//     Enc/Inputs/In/nState2 @bit 1 <-> ENC Status compact/Status/Status of input B
//     Enc/Inputs/In/nState2 @bit 2 <-> ENC Status compact/Status/Status of input C
//     Enc/Inputs/In/nState2 @bit 5 <-> ENC Status compact/Status/Sync error
//     Enc/Inputs/In/nState2 @bit 7 <-> ENC Status compact/Status/TxPDO Toggle
//     Enc/Inputs/In/nState4 @bit 1 <-> WcState/InputToggle
//     Enc/Inputs/In/nState4 <-> WcState/WcState
//     Enc/Outputs/Out/nCtrl1 <-> ENC Control compact/Control/Enable latch C
//     Enc/Outputs/Out/nCtrl1 @bit 3 <-> ENC Control compact/Control/Enable latch extern on negative edge
//     Enc/Outputs/Out/nCtrl1 @bit 1 <-> ENC Control compact/Control/Enable latch extern on positive edge
//     Enc/Outputs/Out/nCtrl1 @bit 2 <-> ENC Control compact/Control/Set counter
//     Enc/Outputs/Out/nDataOut1[0] <-> ENC Control compact/Set counter value
//   (this object) <-> Device 1 (EtherCAT)/Term 5 (EK1200)/Term 6 (EK1122-0080)/DRL02-EK0 (EK1101-0080)/DRL02-E21 (EL7041)
//     Drive/Inputs/In/nState1 @bit 3 <-> STM Status/Status/Error
//     Drive/Inputs/In/nState1 @bit 5 <-> STM Status/Status/Moving negative
//     Drive/Inputs/In/nState1 @bit 4 <-> STM Status/Status/Moving positive
//     Drive/Inputs/In/nState1 @bit 1 <-> STM Status/Status/Ready
//     Drive/Inputs/In/nState1 <-> STM Status/Status/Ready to enable
//     Drive/Inputs/In/nState1 @bit 6 <-> STM Status/Status/Torque reduced
//     Drive/Inputs/In/nState1 @bit 2 <-> STM Status/Status/Warning
//     Drive/Inputs/In/nState2 @bit 3 <-> STM Status/Status/Digital input 1
//     Drive/Inputs/In/nState2 @bit 4 <-> STM Status/Status/Digital input 2
//     Drive/Inputs/In/nState2 @bit 5 <-> STM Status/Status/Sync error
//     Drive/Inputs/In/nState2 @bit 7 <-> STM Status/Status/TxPDO Toggle
//     Drive/Inputs/In/nState4 @bit 1 <-> WcState/InputToggle
//     Drive/Inputs/In/nState4 <-> WcState/WcState
//     Drive/Outputs/Out/nCtrl1 <-> STM Control/Control/Enable
//     Drive/Outputs/Out/nCtrl1 @bit 2 <-> STM Control/Control/Reduce torque
//     Drive/Outputs/Out/nCtrl1 @bit 1 <-> STM Control/Control/Reset
//     Drive/Outputs/Out/nDataOut2[0] <-> STM Velocity/Velocity
//     Enc/Inputs/In/nDataIn1[0] <-> ENC Status compact/Counter value
//     Enc/Inputs/In/nDataIn2[0] <-> ENC Status compact/Latch value
//     Enc/Inputs/In/nState1 @bit 4 <-> ENC Status compact/Status/Counter overflow
//     Enc/Inputs/In/nState1 @bit 3 <-> ENC Status compact/Status/Counter underflow
//     Enc/Inputs/In/nState1 @bit 7 <-> ENC Status compact/Status/Extrapolation stall
//     Enc/Inputs/In/nState1 <-> ENC Status compact/Status/Latch C valid
//     Enc/Inputs/In/nState1 @bit 1 <-> ENC Status compact/Status/Latch extern valid
//     Enc/Inputs/In/nState1 @bit 2 <-> ENC Status compact/Status/Set counter done
//     Enc/Inputs/In/nState2 @bit 4 <-> ENC Status compact/Status/Status of extern latch
//     Enc/Inputs/In/nState2 <-> ENC Status compact/Status/Status of input A
//     Enc/Inputs/In/nState2 @bit 1 <-> ENC Status compact/Status/Status of input B
//     Enc/Inputs/In/nState2 @bit 2 <-> ENC Status compact/Status/Status of input C
//     Enc/Inputs/In/nState2 @bit 5 <-> ENC Status compact/Status/Sync error
//     Enc/Inputs/In/nState2 @bit 7 <-> ENC Status compact/Status/TxPDO Toggle
//     Enc/Inputs/In/nState4 @bit 1 <-> WcState/InputToggle
//     Enc/Inputs/In/nState4 <-> WcState/WcState
//     Enc/Outputs/Out/nCtrl1 <-> ENC Control compact/Control/Enable latch C
//     Enc/Outputs/Out/nCtrl1 @bit 3 <-> ENC Control compact/Control/Enable latch extern on negative edge
//     Enc/Outputs/Out/nCtrl1 @bit 1 <-> ENC Control compact/Control/Enable latch extern on positive edge
//     Enc/Outputs/Out/nCtrl1 @bit 2 <-> ENC Control compact/Control/Set counter
//     Enc/Outputs/Out/nDataOut1[0] <-> ENC Control compact/Set counter value
//   (this object) <-> Device 1 (EtherCAT)/Term 5 (EK1200)/Term 6 (EK1122-0080)/DRL02-EK0 (EK1101-0080)/DRL02-E1 (EL7031)
//     Drive/Inputs/In/nState1 @bit 3 <-> STM Status/Status/Error
//     Drive/Inputs/In/nState1 @bit 5 <-> STM Status/Status/Moving negative
//     Drive/Inputs/In/nState1 @bit 4 <-> STM Status/Status/Moving positive
//     Drive/Inputs/In/nState1 @bit 1 <-> STM Status/Status/Ready
//     Drive/Inputs/In/nState1 <-> STM Status/Status/Ready to enable
//     Drive/Inputs/In/nState1 @bit 6 <-> STM Status/Status/Torque reduced
//     Drive/Inputs/In/nState1 @bit 2 <-> STM Status/Status/Warning
//     Drive/Inputs/In/nState2 @bit 3 <-> STM Status/Status/Digital input 1
//     Drive/Inputs/In/nState2 @bit 4 <-> STM Status/Status/Digital input 2
//     Drive/Inputs/In/nState2 @bit 5 <-> STM Status/Status/Sync error
//     Drive/Inputs/In/nState2 @bit 7 <-> STM Status/Status/TxPDO Toggle
//     Drive/Inputs/In/nState4 @bit 1 <-> WcState/InputToggle
//     Drive/Inputs/In/nState4 <-> WcState/WcState
//     Drive/Outputs/Out/nCtrl1 <-> STM Control/Control/Enable
//     Drive/Outputs/Out/nCtrl1 @bit 2 <-> STM Control/Control/Reduce torque
//     Drive/Outputs/Out/nCtrl1 @bit 1 <-> STM Control/Control/Reset
//     Drive/Outputs/Out/nDataOut2[0] <-> STM Velocity/Velocity
//   (this object) <-> Device 1 (EtherCAT)/Term 5 (EK1200)/Term 6 (EK1122-0080)/DRL02-EK0 (EK1101-0080)/DRL02-E2 (EL5042)
//     Enc/Inputs/In/nComState @bit 1 <-> WcState/InputToggle
//     Enc/Inputs/In/nComState <-> WcState/WcState
//     Enc/Inputs/In/nDataIn1 <-> FB Inputs Channel 1/Position
//     Enc/Inputs/In/nDataIn1 <-> FB Inputs Channel 2/Position
//     Enc/Inputs/In/nState1 @bit 12 <-> FB Inputs Channel 1/Status/Diag
//     Enc/Inputs/In/nState1 @bit 12 <-> FB Inputs Channel 2/Status/Diag
//     Enc/Inputs/In/nState1 @bit 1 <-> FB Inputs Channel 1/Status/Error
//     Enc/Inputs/In/nState1 @bit 1 <-> FB Inputs Channel 2/Status/Error
//     Enc/Inputs/In/nState1 @bit 14 <-> FB Inputs Channel 1/Status/Input cycle counter
//     Enc/Inputs/In/nState1 @bit 14 <-> FB Inputs Channel 2/Status/Input cycle counter
//     Enc/Inputs/In/nState1 @bit 2 <-> FB Inputs Channel 1/Status/Ready
//     Enc/Inputs/In/nState1 @bit 2 <-> FB Inputs Channel 2/Status/Ready
//     Enc/Inputs/In/nState1 @bit 13 <-> FB Inputs Channel 1/Status/TxPDO State
//     Enc/Inputs/In/nState1 @bit 13 <-> FB Inputs Channel 2/Status/TxPDO State
//     Enc/Inputs/In/nState1 <-> FB Inputs Channel 1/Status/Warning
//     Enc/Inputs/In/nState1 <-> FB Inputs Channel 2/Status/Warning
//   (this object) <-> Device 1 (EtherCAT)/Term 5 (EK1200)/Term 6 (EK1122-0080)/DRL02-EK0 (EK1101-0080)/DRL02-E3 (EL7031)
//     Drive/Inputs/In/nState1 @bit 3 <-> STM Status/Status/Error
//     Drive/Inputs/In/nState1 @bit 5 <-> STM Status/Status/Moving negative
//     Drive/Inputs/In/nState1 @bit 4 <-> STM Status/Status/Moving positive
//     Drive/Inputs/In/nState1 @bit 1 <-> STM Status/Status/Ready
//     Drive/Inputs/In/nState1 <-> STM Status/Status/Ready to enable
//     Drive/Inputs/In/nState1 @bit 6 <-> STM Status/Status/Torque reduced
//     Drive/Inputs/In/nState1 @bit 2 <-> STM Status/Status/Warning
//     Drive/Inputs/In/nState2 @bit 3 <-> STM Status/Status/Digital input 1
//     Drive/Inputs/In/nState2 @bit 4 <-> STM Status/Status/Digital input 2
//     Drive/Inputs/In/nState2 @bit 5 <-> STM Status/Status/Sync error
//     Drive/Inputs/In/nState2 @bit 7 <-> STM Status/Status/TxPDO Toggle
//     Drive/Inputs/In/nState4 @bit 1 <-> WcState/InputToggle
//     Drive/Inputs/In/nState4 <-> WcState/WcState
//     Drive/Outputs/Out/nCtrl1 <-> STM Control/Control/Enable
//     Drive/Outputs/Out/nCtrl1 @bit 2 <-> STM Control/Control/Reduce torque
//     Drive/Outputs/Out/nCtrl1 @bit 1 <-> STM Control/Control/Reset
//     Drive/Outputs/Out/nDataOut2[0] <-> STM Velocity/Velocity
//   (this object) <-> Device 1 (EtherCAT)/Term 5 (EK1200)/Term 6 (EK1122-0080)/DRL02-EK0 (EK1101-0080)/DRL02-E4 (EL7031)
//     Drive/Inputs/In/nState1 @bit 3 <-> STM Status/Status/Error
//     Drive/Inputs/In/nState1 @bit 5 <-> STM Status/Status/Moving negative
//     Drive/Inputs/In/nState1 @bit 4 <-> STM Status/Status/Moving positive
//     Drive/Inputs/In/nState1 @bit 1 <-> STM Status/Status/Ready
//     Drive/Inputs/In/nState1 <-> STM Status/Status/Ready to enable
//     Drive/Inputs/In/nState1 @bit 6 <-> STM Status/Status/Torque reduced
//     Drive/Inputs/In/nState1 @bit 2 <-> STM Status/Status/Warning
//     Drive/Inputs/In/nState2 @bit 3 <-> STM Status/Status/Digital input 1
//     Drive/Inputs/In/nState2 @bit 4 <-> STM Status/Status/Digital input 2
//     Drive/Inputs/In/nState2 @bit 5 <-> STM Status/Status/Sync error
//     Drive/Inputs/In/nState2 @bit 7 <-> STM Status/Status/TxPDO Toggle
//     Drive/Inputs/In/nState4 @bit 1 <-> WcState/InputToggle
//     Drive/Inputs/In/nState4 <-> WcState/WcState
//     Drive/Outputs/Out/nCtrl1 <-> STM Control/Control/Enable
//     Drive/Outputs/Out/nCtrl1 @bit 2 <-> STM Control/Control/Reduce torque
//     Drive/Outputs/Out/nCtrl1 @bit 1 <-> STM Control/Control/Reset
//     Drive/Outputs/Out/nDataOut2[0] <-> STM Velocity/Velocity
//   (this object) <-> Device 1 (EtherCAT)/Term 5 (EK1200)/Term 6 (EK1122-0080)/DRL02-EK0 (EK1101-0080)/DRL02-E5 (EL5042)
//     Enc/Inputs/In/nComState @bit 1 <-> WcState/InputToggle
//     Enc/Inputs/In/nComState <-> WcState/WcState
//     Enc/Inputs/In/nDataIn1 <-> FB Inputs Channel 1/Position
//     Enc/Inputs/In/nDataIn1 <-> FB Inputs Channel 2/Position
//     Enc/Inputs/In/nState1 @bit 12 <-> FB Inputs Channel 1/Status/Diag
//     Enc/Inputs/In/nState1 @bit 12 <-> FB Inputs Channel 2/Status/Diag
//     Enc/Inputs/In/nState1 @bit 1 <-> FB Inputs Channel 1/Status/Error
//     Enc/Inputs/In/nState1 @bit 1 <-> FB Inputs Channel 2/Status/Error
//     Enc/Inputs/In/nState1 @bit 14 <-> FB Inputs Channel 1/Status/Input cycle counter
//     Enc/Inputs/In/nState1 @bit 14 <-> FB Inputs Channel 2/Status/Input cycle counter
//     Enc/Inputs/In/nState1 @bit 2 <-> FB Inputs Channel 1/Status/Ready
//     Enc/Inputs/In/nState1 @bit 2 <-> FB Inputs Channel 2/Status/Ready
//     Enc/Inputs/In/nState1 @bit 13 <-> FB Inputs Channel 1/Status/TxPDO State
//     Enc/Inputs/In/nState1 @bit 13 <-> FB Inputs Channel 2/Status/TxPDO State
//     Enc/Inputs/In/nState1 <-> FB Inputs Channel 1/Status/Warning
//     Enc/Inputs/In/nState1 <-> FB Inputs Channel 2/Status/Warning
//   (this object) <-> Device 1 (EtherCAT)/Term 5 (EK1200)/Term 6 (EK1122-0080)/DRL02-EK0 (EK1101-0080)/DRL02-E6 (EL7031)
//     Drive/Inputs/In/nState1 @bit 3 <-> STM Status/Status/Error
//     Drive/Inputs/In/nState1 @bit 5 <-> STM Status/Status/Moving negative
//     Drive/Inputs/In/nState1 @bit 4 <-> STM Status/Status/Moving positive
//     Drive/Inputs/In/nState1 @bit 1 <-> STM Status/Status/Ready
//     Drive/Inputs/In/nState1 <-> STM Status/Status/Ready to enable
//     Drive/Inputs/In/nState1 @bit 6 <-> STM Status/Status/Torque reduced
//     Drive/Inputs/In/nState1 @bit 2 <-> STM Status/Status/Warning
//     Drive/Inputs/In/nState2 @bit 3 <-> STM Status/Status/Digital input 1
//     Drive/Inputs/In/nState2 @bit 4 <-> STM Status/Status/Digital input 2
//     Drive/Inputs/In/nState2 @bit 5 <-> STM Status/Status/Sync error
//     Drive/Inputs/In/nState2 @bit 7 <-> STM Status/Status/TxPDO Toggle
//     Drive/Inputs/In/nState4 @bit 1 <-> WcState/InputToggle
//     Drive/Inputs/In/nState4 <-> WcState/WcState
//     Drive/Outputs/Out/nCtrl1 <-> STM Control/Control/Enable
//     Drive/Outputs/Out/nCtrl1 @bit 2 <-> STM Control/Control/Reduce torque
//     Drive/Outputs/Out/nCtrl1 @bit 1 <-> STM Control/Control/Reset
//     Drive/Outputs/Out/nDataOut2[0] <-> STM Velocity/Velocity
//   (this object) <-> Device 1 (EtherCAT)/Term 5 (EK1200)/Term 6 (EK1122-0080)/DRL02-EK0 (EK1101-0080)/DRL02-E7 (EL7031)
//     Drive/Inputs/In/nState1 @bit 3 <-> STM Status/Status/Error
//     Drive/Inputs/In/nState1 @bit 5 <-> STM Status/Status/Moving negative
//     Drive/Inputs/In/nState1 @bit 4 <-> STM Status/Status/Moving positive
//     Drive/Inputs/In/nState1 @bit 1 <-> STM Status/Status/Ready
//     Drive/Inputs/In/nState1 <-> STM Status/Status/Ready to enable
//     Drive/Inputs/In/nState1 @bit 6 <-> STM Status/Status/Torque reduced
//     Drive/Inputs/In/nState1 @bit 2 <-> STM Status/Status/Warning
//     Drive/Inputs/In/nState2 @bit 3 <-> STM Status/Status/Digital input 1
//     Drive/Inputs/In/nState2 @bit 4 <-> STM Status/Status/Digital input 2
//     Drive/Inputs/In/nState2 @bit 5 <-> STM Status/Status/Sync error
//     Drive/Inputs/In/nState2 @bit 7 <-> STM Status/Status/TxPDO Toggle
//     Drive/Inputs/In/nState4 @bit 1 <-> WcState/InputToggle
//     Drive/Inputs/In/nState4 <-> WcState/WcState
//     Drive/Outputs/Out/nCtrl1 <-> STM Control/Control/Enable
//     Drive/Outputs/Out/nCtrl1 @bit 2 <-> STM Control/Control/Reduce torque
//     Drive/Outputs/Out/nCtrl1 @bit 1 <-> STM Control/Control/Reset
//     Drive/Outputs/Out/nDataOut2[0] <-> STM Velocity/Velocity
//   (this object) <-> Device 1 (EtherCAT)/Term 5 (EK1200)/Term 6 (EK1122-0080)/DRL02-EK0 (EK1101-0080)/DRL02-E8 (EL5042)
//     Enc/Inputs/In/nComState @bit 1 <-> WcState/InputToggle
//     Enc/Inputs/In/nComState <-> WcState/WcState
//     Enc/Inputs/In/nDataIn1 <-> FB Inputs Channel 1/Position
//     Enc/Inputs/In/nDataIn1 <-> FB Inputs Channel 2/Position
//     Enc/Inputs/In/nState1 @bit 12 <-> FB Inputs Channel 1/Status/Diag
//     Enc/Inputs/In/nState1 @bit 12 <-> FB Inputs Channel 2/Status/Diag
//     Enc/Inputs/In/nState1 @bit 1 <-> FB Inputs Channel 1/Status/Error
//     Enc/Inputs/In/nState1 @bit 1 <-> FB Inputs Channel 2/Status/Error
//     Enc/Inputs/In/nState1 @bit 14 <-> FB Inputs Channel 1/Status/Input cycle counter
//     Enc/Inputs/In/nState1 @bit 14 <-> FB Inputs Channel 2/Status/Input cycle counter
//     Enc/Inputs/In/nState1 @bit 2 <-> FB Inputs Channel 1/Status/Ready
//     Enc/Inputs/In/nState1 @bit 2 <-> FB Inputs Channel 2/Status/Ready
//     Enc/Inputs/In/nState1 @bit 13 <-> FB Inputs Channel 1/Status/TxPDO State
//     Enc/Inputs/In/nState1 @bit 13 <-> FB Inputs Channel 2/Status/TxPDO State
//     Enc/Inputs/In/nState1 <-> FB Inputs Channel 1/Status/Warning
//     Enc/Inputs/In/nState1 <-> FB Inputs Channel 2/Status/Warning
//   (this object) <-> Device 1 (EtherCAT)/Term 5 (EK1200)/Term 6 (EK1122-0080)/DRL02-EK0 (EK1101-0080)/DRL02-E9 (EL7031)
//     Drive/Inputs/In/nState1 @bit 3 <-> STM Status/Status/Error
//     Drive/Inputs/In/nState1 @bit 5 <-> STM Status/Status/Moving negative
//     Drive/Inputs/In/nState1 @bit 4 <-> STM Status/Status/Moving positive
//     Drive/Inputs/In/nState1 @bit 1 <-> STM Status/Status/Ready
//     Drive/Inputs/In/nState1 <-> STM Status/Status/Ready to enable
//     Drive/Inputs/In/nState1 @bit 6 <-> STM Status/Status/Torque reduced
//     Drive/Inputs/In/nState1 @bit 2 <-> STM Status/Status/Warning
//     Drive/Inputs/In/nState2 @bit 3 <-> STM Status/Status/Digital input 1
//     Drive/Inputs/In/nState2 @bit 4 <-> STM Status/Status/Digital input 2
//     Drive/Inputs/In/nState2 @bit 5 <-> STM Status/Status/Sync error
//     Drive/Inputs/In/nState2 @bit 7 <-> STM Status/Status/TxPDO Toggle
//     Drive/Inputs/In/nState4 @bit 1 <-> WcState/InputToggle
//     Drive/Inputs/In/nState4 <-> WcState/WcState
//     Drive/Outputs/Out/nCtrl1 <-> STM Control/Control/Enable
//     Drive/Outputs/Out/nCtrl1 @bit 2 <-> STM Control/Control/Reduce torque
//     Drive/Outputs/Out/nCtrl1 @bit 1 <-> STM Control/Control/Reset
//     Drive/Outputs/Out/nDataOut2[0] <-> STM Velocity/Velocity
//   (this object) <-> Device 1 (EtherCAT)/Term 5 (EK1200)/Term 6 (EK1122-0080)/DRL02-EK0 (EK1101-0080)/DRL02-E11 (EL7031)
//     Drive/Inputs/In/nState1 @bit 3 <-> STM Status/Status/Error
//     Drive/Inputs/In/nState1 @bit 5 <-> STM Status/Status/Moving negative
//     Drive/Inputs/In/nState1 @bit 4 <-> STM Status/Status/Moving positive
//     Drive/Inputs/In/nState1 @bit 1 <-> STM Status/Status/Ready
//     Drive/Inputs/In/nState1 <-> STM Status/Status/Ready to enable
//     Drive/Inputs/In/nState1 @bit 6 <-> STM Status/Status/Torque reduced
//     Drive/Inputs/In/nState1 @bit 2 <-> STM Status/Status/Warning
//     Drive/Inputs/In/nState2 @bit 3 <-> STM Status/Status/Digital input 1
//     Drive/Inputs/In/nState2 @bit 4 <-> STM Status/Status/Digital input 2
//     Drive/Inputs/In/nState2 @bit 5 <-> STM Status/Status/Sync error
//     Drive/Inputs/In/nState2 @bit 7 <-> STM Status/Status/TxPDO Toggle
//     Drive/Inputs/In/nState4 @bit 1 <-> WcState/InputToggle
//     Drive/Inputs/In/nState4 <-> WcState/WcState
//     Drive/Outputs/Out/nCtrl1 <-> STM Control/Control/Enable
//     Drive/Outputs/Out/nCtrl1 @bit 2 <-> STM Control/Control/Reduce torque
//     Drive/Outputs/Out/nCtrl1 @bit 1 <-> STM Control/Control/Reset
//     Drive/Outputs/Out/nDataOut2[0] <-> STM Velocity/Velocity
//   (this object) <-> Device 1 (EtherCAT)/Term 5 (EK1200)/Term 6 (EK1122-0080)/DRL02-EK0 (EK1101-0080)/DRL02-E12 (EL5042)
//     Enc/Inputs/In/nComState @bit 1 <-> WcState/InputToggle
//     Enc/Inputs/In/nComState <-> WcState/WcState
//     Enc/Inputs/In/nDataIn1 <-> FB Inputs Channel 1/Position
//     Enc/Inputs/In/nDataIn1 <-> FB Inputs Channel 2/Position
//     Enc/Inputs/In/nState1 @bit 12 <-> FB Inputs Channel 1/Status/Diag
//     Enc/Inputs/In/nState1 @bit 12 <-> FB Inputs Channel 2/Status/Diag
//     Enc/Inputs/In/nState1 @bit 1 <-> FB Inputs Channel 1/Status/Error
//     Enc/Inputs/In/nState1 @bit 1 <-> FB Inputs Channel 2/Status/Error
//     Enc/Inputs/In/nState1 @bit 14 <-> FB Inputs Channel 1/Status/Input cycle counter
//     Enc/Inputs/In/nState1 @bit 14 <-> FB Inputs Channel 2/Status/Input cycle counter
//     Enc/Inputs/In/nState1 @bit 2 <-> FB Inputs Channel 1/Status/Ready
//     Enc/Inputs/In/nState1 @bit 2 <-> FB Inputs Channel 2/Status/Ready
//     Enc/Inputs/In/nState1 @bit 13 <-> FB Inputs Channel 1/Status/TxPDO State
//     Enc/Inputs/In/nState1 @bit 13 <-> FB Inputs Channel 2/Status/TxPDO State
//     Enc/Inputs/In/nState1 <-> FB Inputs Channel 1/Status/Warning
//     Enc/Inputs/In/nState1 <-> FB Inputs Channel 2/Status/Warning
//   (this object) <-> Device 1 (EtherCAT)/Term 5 (EK1200)/Term 6 (EK1122-0080)/DRL02-EK0 (EK1101-0080)/DRL02-E13 (EL7041)
//     Drive/Inputs/In/nState1 @bit 3 <-> STM Status/Status/Error
//     Drive/Inputs/In/nState1 @bit 5 <-> STM Status/Status/Moving negative
//     Drive/Inputs/In/nState1 @bit 4 <-> STM Status/Status/Moving positive
//     Drive/Inputs/In/nState1 @bit 1 <-> STM Status/Status/Ready
//     Drive/Inputs/In/nState1 <-> STM Status/Status/Ready to enable
//     Drive/Inputs/In/nState1 @bit 6 <-> STM Status/Status/Torque reduced
//     Drive/Inputs/In/nState1 @bit 2 <-> STM Status/Status/Warning
//     Drive/Inputs/In/nState2 @bit 3 <-> STM Status/Status/Digital input 1
//     Drive/Inputs/In/nState2 @bit 4 <-> STM Status/Status/Digital input 2
//     Drive/Inputs/In/nState2 @bit 5 <-> STM Status/Status/Sync error
//     Drive/Inputs/In/nState2 @bit 7 <-> STM Status/Status/TxPDO Toggle
//     Drive/Inputs/In/nState4 @bit 1 <-> WcState/InputToggle
//     Drive/Inputs/In/nState4 <-> WcState/WcState
//     Drive/Outputs/Out/nCtrl1 <-> STM Control/Control/Enable
//     Drive/Outputs/Out/nCtrl1 @bit 2 <-> STM Control/Control/Reduce torque
//     Drive/Outputs/Out/nCtrl1 @bit 1 <-> STM Control/Control/Reset
//     Drive/Outputs/Out/nDataOut2[0] <-> STM Velocity/Velocity
//   (this object) <-> Device 1 (EtherCAT)/Term 5 (EK1200)/Term 6 (EK1122-0080)/DRL02-EK0 (EK1101-0080)/DRL02-E14 (EL7041)
//     Drive/Inputs/In/nState1 @bit 3 <-> STM Status/Status/Error
//     Drive/Inputs/In/nState1 @bit 5 <-> STM Status/Status/Moving negative
//     Drive/Inputs/In/nState1 @bit 4 <-> STM Status/Status/Moving positive
//     Drive/Inputs/In/nState1 @bit 1 <-> STM Status/Status/Ready
//     Drive/Inputs/In/nState1 <-> STM Status/Status/Ready to enable
//     Drive/Inputs/In/nState1 @bit 6 <-> STM Status/Status/Torque reduced
//     Drive/Inputs/In/nState1 @bit 2 <-> STM Status/Status/Warning
//     Drive/Inputs/In/nState2 @bit 3 <-> STM Status/Status/Digital input 1
//     Drive/Inputs/In/nState2 @bit 4 <-> STM Status/Status/Digital input 2
//     Drive/Inputs/In/nState2 @bit 5 <-> STM Status/Status/Sync error
//     Drive/Inputs/In/nState2 @bit 7 <-> STM Status/Status/TxPDO Toggle
//     Drive/Inputs/In/nState4 @bit 1 <-> WcState/InputToggle
//     Drive/Inputs/In/nState4 <-> WcState/WcState
//     Drive/Outputs/Out/nCtrl1 <-> STM Control/Control/Enable
//     Drive/Outputs/Out/nCtrl1 @bit 2 <-> STM Control/Control/Reduce torque
//     Drive/Outputs/Out/nCtrl1 @bit 1 <-> STM Control/Control/Reset
//     Drive/Outputs/Out/nDataOut2[0] <-> STM Velocity/Velocity
//     Enc/Inputs/In/nDataIn1[0] <-> ENC Status compact/Counter value
//     Enc/Inputs/In/nDataIn2[0] <-> ENC Status compact/Latch value
//     Enc/Inputs/In/nState1 @bit 4 <-> ENC Status compact/Status/Counter overflow
//     Enc/Inputs/In/nState1 @bit 3 <-> ENC Status compact/Status/Counter underflow
//     Enc/Inputs/In/nState1 @bit 7 <-> ENC Status compact/Status/Extrapolation stall
//     Enc/Inputs/In/nState1 <-> ENC Status compact/Status/Latch C valid
//     Enc/Inputs/In/nState1 @bit 1 <-> ENC Status compact/Status/Latch extern valid
//     Enc/Inputs/In/nState1 @bit 2 <-> ENC Status compact/Status/Set counter done
//     Enc/Inputs/In/nState2 @bit 4 <-> ENC Status compact/Status/Status of extern latch
//     Enc/Inputs/In/nState2 <-> ENC Status compact/Status/Status of input A
//     Enc/Inputs/In/nState2 @bit 1 <-> ENC Status compact/Status/Status of input B
//     Enc/Inputs/In/nState2 @bit 2 <-> ENC Status compact/Status/Status of input C
//     Enc/Inputs/In/nState2 @bit 5 <-> ENC Status compact/Status/Sync error
//     Enc/Inputs/In/nState2 @bit 7 <-> ENC Status compact/Status/TxPDO Toggle
//     Enc/Inputs/In/nState4 @bit 1 <-> WcState/InputToggle
//     Enc/Inputs/In/nState4 <-> WcState/WcState
//     Enc/Outputs/Out/nCtrl1 <-> ENC Control compact/Control/Enable latch C
//     Enc/Outputs/Out/nCtrl1 @bit 3 <-> ENC Control compact/Control/Enable latch extern on negative edge
//     Enc/Outputs/Out/nCtrl1 @bit 1 <-> ENC Control compact/Control/Enable latch extern on positive edge
//     Enc/Outputs/Out/nCtrl1 @bit 2 <-> ENC Control compact/Control/Set counter
//     Enc/Outputs/Out/nDataOut1[0] <-> ENC Control compact/Set counter value
//   (this object) <-> Device 1 (EtherCAT)/Term 5 (EK1200)/Term 6 (EK1122-0080)/DRL02-EK0 (EK1101-0080)/Term 66 (EL7031)
//     Drive/Inputs/In/nState1 @bit 3 <-> STM Status/Status/Error
//     Drive/Inputs/In/nState1 @bit 5 <-> STM Status/Status/Moving negative
//     Drive/Inputs/In/nState1 @bit 4 <-> STM Status/Status/Moving positive
//     Drive/Inputs/In/nState1 @bit 1 <-> STM Status/Status/Ready
//     Drive/Inputs/In/nState1 <-> STM Status/Status/Ready to enable
//     Drive/Inputs/In/nState1 @bit 6 <-> STM Status/Status/Torque reduced
//     Drive/Inputs/In/nState1 @bit 2 <-> STM Status/Status/Warning
//     Drive/Inputs/In/nState2 @bit 3 <-> STM Status/Status/Digital input 1
//     Drive/Inputs/In/nState2 @bit 4 <-> STM Status/Status/Digital input 2
//     Drive/Inputs/In/nState2 @bit 5 <-> STM Status/Status/Sync error
//     Drive/Inputs/In/nState2 @bit 7 <-> STM Status/Status/TxPDO Toggle
//     Drive/Inputs/In/nState4 @bit 1 <-> WcState/InputToggle
//     Drive/Inputs/In/nState4 <-> WcState/WcState
//     Drive/Outputs/Out/nCtrl1 <-> STM Control/Control/Enable
//     Drive/Outputs/Out/nCtrl1 @bit 2 <-> STM Control/Control/Reduce torque
//     Drive/Outputs/Out/nCtrl1 @bit 1 <-> STM Control/Control/Reset
//     Drive/Outputs/Out/nDataOut2[0] <-> STM Velocity/Velocity
//     Enc/Inputs/In/nDataIn1[0] <-> ENC Status compact/Counter value
//     Enc/Inputs/In/nDataIn2[0] <-> ENC Status compact/Latch value
//     Enc/Inputs/In/nState1 @bit 4 <-> ENC Status compact/Status/Counter overflow
//     Enc/Inputs/In/nState1 @bit 3 <-> ENC Status compact/Status/Counter underflow
//     Enc/Inputs/In/nState1 @bit 1 <-> ENC Status compact/Status/Latch extern valid
//     Enc/Inputs/In/nState1 @bit 2 <-> ENC Status compact/Status/Set counter done
//     Enc/Inputs/In/nState2 @bit 4 <-> ENC Status compact/Status/Status of extern latch
//     Enc/Inputs/In/nState2 @bit 5 <-> ENC Status compact/Status/Sync error
//     Enc/Inputs/In/nState2 @bit 7 <-> ENC Status compact/Status/TxPDO Toggle
//     Enc/Inputs/In/nState4 @bit 1 <-> WcState/InputToggle
//     Enc/Inputs/In/nState4 <-> WcState/WcState
//     Enc/Outputs/Out/nCtrl1 @bit 3 <-> ENC Control compact/Control/Enable latch extern on negative edge
//     Enc/Outputs/Out/nCtrl1 @bit 1 <-> ENC Control compact/Control/Enable latch extern on positive edge
//     Enc/Outputs/Out/nCtrl1 @bit 2 <-> ENC Control compact/Control/Set counter
//     Enc/Outputs/Out/nDataOut1[0] <-> ENC Control compact/Set counter value
//   (this object) <-> Device 1 (EtherCAT)/Term 5 (EK1200)/Term 6 (EK1122-0080)/DRL02-EK0 (EK1101-0080)/DRL02-E16 (EL7041)
//     Drive/Inputs/In/nState1 @bit 3 <-> STM Status/Status/Error
//     Drive/Inputs/In/nState1 @bit 5 <-> STM Status/Status/Moving negative
//     Drive/Inputs/In/nState1 @bit 4 <-> STM Status/Status/Moving positive
//     Drive/Inputs/In/nState1 @bit 1 <-> STM Status/Status/Ready
//     Drive/Inputs/In/nState1 <-> STM Status/Status/Ready to enable
//     Drive/Inputs/In/nState1 @bit 6 <-> STM Status/Status/Torque reduced
//     Drive/Inputs/In/nState1 @bit 2 <-> STM Status/Status/Warning
//     Drive/Inputs/In/nState2 @bit 3 <-> STM Status/Status/Digital input 1
//     Drive/Inputs/In/nState2 @bit 4 <-> STM Status/Status/Digital input 2
//     Drive/Inputs/In/nState2 @bit 5 <-> STM Status/Status/Sync error
//     Drive/Inputs/In/nState2 @bit 7 <-> STM Status/Status/TxPDO Toggle
//     Drive/Inputs/In/nState4 @bit 1 <-> WcState/InputToggle
//     Drive/Inputs/In/nState4 <-> WcState/WcState
//     Drive/Outputs/Out/nCtrl1 <-> STM Control/Control/Enable
//     Drive/Outputs/Out/nCtrl1 @bit 2 <-> STM Control/Control/Reduce torque
//     Drive/Outputs/Out/nCtrl1 @bit 1 <-> STM Control/Control/Reset
//     Drive/Outputs/Out/nDataOut2[0] <-> STM Velocity/Velocity
//     Enc/Inputs/In/nDataIn1[0] <-> ENC Status compact/Counter value
//     Enc/Inputs/In/nDataIn2[0] <-> ENC Status compact/Latch value
//     Enc/Inputs/In/nState1 @bit 4 <-> ENC Status compact/Status/Counter overflow
//     Enc/Inputs/In/nState1 @bit 3 <-> ENC Status compact/Status/Counter underflow
//     Enc/Inputs/In/nState1 @bit 7 <-> ENC Status compact/Status/Extrapolation stall
//     Enc/Inputs/In/nState1 <-> ENC Status compact/Status/Latch C valid
//     Enc/Inputs/In/nState1 @bit 1 <-> ENC Status compact/Status/Latch extern valid
//     Enc/Inputs/In/nState1 @bit 2 <-> ENC Status compact/Status/Set counter done
//     Enc/Inputs/In/nState2 @bit 4 <-> ENC Status compact/Status/Status of extern latch
//     Enc/Inputs/In/nState2 <-> ENC Status compact/Status/Status of input A
//     Enc/Inputs/In/nState2 @bit 1 <-> ENC Status compact/Status/Status of input B
//     Enc/Inputs/In/nState2 @bit 2 <-> ENC Status compact/Status/Status of input C
//     Enc/Inputs/In/nState2 @bit 5 <-> ENC Status compact/Status/Sync error
//     Enc/Inputs/In/nState2 @bit 7 <-> ENC Status compact/Status/TxPDO Toggle
//     Enc/Inputs/In/nState4 @bit 1 <-> WcState/InputToggle
//     Enc/Inputs/In/nState4 <-> WcState/WcState
//     Enc/Outputs/Out/nCtrl1 <-> ENC Control compact/Control/Enable latch C
//     Enc/Outputs/Out/nCtrl1 @bit 3 <-> ENC Control compact/Control/Enable latch extern on negative edge
//     Enc/Outputs/Out/nCtrl1 @bit 1 <-> ENC Control compact/Control/Enable latch extern on positive edge
//     Enc/Outputs/Out/nCtrl1 @bit 2 <-> ENC Control compact/Control/Set counter
//     Enc/Outputs/Out/nDataOut1[0] <-> ENC Control compact/Set counter value
//   (this object) <-> Device 1 (EtherCAT)/Term 5 (EK1200)/Term 6 (EK1122-0080)/DRL02-EK0 (EK1101-0080)/DRL02-E17 (EL7031)
//     Drive/Inputs/In/nState1 @bit 3 <-> STM Status/Status/Error
//     Drive/Inputs/In/nState1 @bit 5 <-> STM Status/Status/Moving negative
//     Drive/Inputs/In/nState1 @bit 4 <-> STM Status/Status/Moving positive
//     Drive/Inputs/In/nState1 @bit 1 <-> STM Status/Status/Ready
//     Drive/Inputs/In/nState1 <-> STM Status/Status/Ready to enable
//     Drive/Inputs/In/nState1 @bit 6 <-> STM Status/Status/Torque reduced
//     Drive/Inputs/In/nState1 @bit 2 <-> STM Status/Status/Warning
//     Drive/Inputs/In/nState2 @bit 3 <-> STM Status/Status/Digital input 1
//     Drive/Inputs/In/nState2 @bit 4 <-> STM Status/Status/Digital input 2
//     Drive/Inputs/In/nState2 @bit 5 <-> STM Status/Status/Sync error
//     Drive/Inputs/In/nState2 @bit 7 <-> STM Status/Status/TxPDO Toggle
//     Drive/Inputs/In/nState4 @bit 1 <-> WcState/InputToggle
//     Drive/Inputs/In/nState4 <-> WcState/WcState
//     Drive/Outputs/Out/nCtrl1 <-> STM Control/Control/Enable
//     Drive/Outputs/Out/nCtrl1 @bit 2 <-> STM Control/Control/Reduce torque
//     Drive/Outputs/Out/nCtrl1 @bit 1 <-> STM Control/Control/Reset
//     Drive/Outputs/Out/nDataOut2[0] <-> STM Velocity/Velocity
//   (this object) <-> Device 1 (EtherCAT)/Term 5 (EK1200)/Term 6 (EK1122-0080)/DRL02-EK0 (EK1101-0080)/DRL02-E18 (EL5042)
//     Enc/Inputs/In/nComState @bit 1 <-> WcState/InputToggle
//     Enc/Inputs/In/nComState <-> WcState/WcState
//     Enc/Inputs/In/nDataIn1 <-> FB Inputs Channel 1/Position
//     Enc/Inputs/In/nDataIn1 <-> FB Inputs Channel 2/Position
//     Enc/Inputs/In/nState1 @bit 12 <-> FB Inputs Channel 1/Status/Diag
//     Enc/Inputs/In/nState1 @bit 12 <-> FB Inputs Channel 2/Status/Diag
//     Enc/Inputs/In/nState1 @bit 1 <-> FB Inputs Channel 1/Status/Error
//     Enc/Inputs/In/nState1 @bit 1 <-> FB Inputs Channel 2/Status/Error
//     Enc/Inputs/In/nState1 @bit 14 <-> FB Inputs Channel 1/Status/Input cycle counter
//     Enc/Inputs/In/nState1 @bit 14 <-> FB Inputs Channel 2/Status/Input cycle counter
//     Enc/Inputs/In/nState1 @bit 2 <-> FB Inputs Channel 1/Status/Ready
//     Enc/Inputs/In/nState1 @bit 2 <-> FB Inputs Channel 2/Status/Ready
//     Enc/Inputs/In/nState1 @bit 13 <-> FB Inputs Channel 1/Status/TxPDO State
//     Enc/Inputs/In/nState1 @bit 13 <-> FB Inputs Channel 2/Status/TxPDO State
//     Enc/Inputs/In/nState1 <-> FB Inputs Channel 1/Status/Warning
//     Enc/Inputs/In/nState1 <-> FB Inputs Channel 2/Status/Warning
//   (this object) <-> Device 1 (EtherCAT)/Term 5 (EK1200)/Term 6 (EK1122-0080)/DRL02-EK0 (EK1101-0080)/DRL02-E19 (EL7031)
//     Drive/Inputs/In/nState1 @bit 3 <-> STM Status/Status/Error
//     Drive/Inputs/In/nState1 @bit 5 <-> STM Status/Status/Moving negative
//     Drive/Inputs/In/nState1 @bit 4 <-> STM Status/Status/Moving positive
//     Drive/Inputs/In/nState1 @bit 1 <-> STM Status/Status/Ready
//     Drive/Inputs/In/nState1 <-> STM Status/Status/Ready to enable
//     Drive/Inputs/In/nState1 @bit 6 <-> STM Status/Status/Torque reduced
//     Drive/Inputs/In/nState1 @bit 2 <-> STM Status/Status/Warning
//     Drive/Inputs/In/nState2 @bit 3 <-> STM Status/Status/Digital input 1
//     Drive/Inputs/In/nState2 @bit 4 <-> STM Status/Status/Digital input 2
//     Drive/Inputs/In/nState2 @bit 5 <-> STM Status/Status/Sync error
//     Drive/Inputs/In/nState2 @bit 7 <-> STM Status/Status/TxPDO Toggle
//     Drive/Inputs/In/nState4 @bit 1 <-> WcState/InputToggle
//     Drive/Inputs/In/nState4 <-> WcState/WcState
//     Drive/Outputs/Out/nCtrl1 <-> STM Control/Control/Enable
//     Drive/Outputs/Out/nCtrl1 @bit 2 <-> STM Control/Control/Reduce torque
//     Drive/Outputs/Out/nCtrl1 @bit 1 <-> STM Control/Control/Reset
//     Drive/Outputs/Out/nDataOut2[0] <-> STM Velocity/Velocity
//   (this object) <-> Device 1 (EtherCAT)/Term 5 (EK1200)/Term 6 (EK1122-0080)/DRL02-EK0 (EK1101-0080)/DRL02-E24 (EL7031)
//     Drive/Inputs/In/nState1 @bit 3 <-> STM Status/Status/Error
//     Drive/Inputs/In/nState1 @bit 5 <-> STM Status/Status/Moving negative
//     Drive/Inputs/In/nState1 @bit 4 <-> STM Status/Status/Moving positive
//     Drive/Inputs/In/nState1 @bit 1 <-> STM Status/Status/Ready
//     Drive/Inputs/In/nState1 <-> STM Status/Status/Ready to enable
//     Drive/Inputs/In/nState1 @bit 6 <-> STM Status/Status/Torque reduced
//     Drive/Inputs/In/nState1 @bit 2 <-> STM Status/Status/Warning
//     Drive/Inputs/In/nState2 @bit 3 <-> STM Status/Status/Digital input 1
//     Drive/Inputs/In/nState2 @bit 4 <-> STM Status/Status/Digital input 2
//     Drive/Inputs/In/nState2 @bit 5 <-> STM Status/Status/Sync error
//     Drive/Inputs/In/nState2 @bit 7 <-> STM Status/Status/TxPDO Toggle
//     Drive/Inputs/In/nState4 @bit 1 <-> WcState/InputToggle
//     Drive/Inputs/In/nState4 <-> WcState/WcState
//     Drive/Outputs/Out/nCtrl1 <-> STM Control/Control/Enable
//     Drive/Outputs/Out/nCtrl1 @bit 2 <-> STM Control/Control/Reduce torque
//     Drive/Outputs/Out/nCtrl1 @bit 1 <-> STM Control/Control/Reset
//     Drive/Outputs/Out/nDataOut2[0] <-> STM Velocity/Velocity
//   (this object) <-> Device 1 (EtherCAT)/Term 5 (EK1200)/Term 6 (EK1122-0080)/DRL02-EK0 (EK1101-0080)/Term 91 (EL5112)
//     Enc/Inputs/In/nDataIn1 <-> ENC Status Channel 1/Counter value
//     Enc/Inputs/In/nDataIn2 <-> ENC Status Channel 1/Latch value
//     Enc/Inputs/In/nState1 @bit 4 <-> ENC Status Channel 1/Status/Counter overflow
//     Enc/Inputs/In/nState1 @bit 3 <-> ENC Status Channel 1/Status/Counter underflow
//     Enc/Inputs/In/nState1 @bit 1 <-> ENC Status Channel 1/Status/Latch extern valid
//     Enc/Inputs/In/nState1 @bit 6 <-> ENC Status Channel 1/Status/Open circuit
//     Enc/Inputs/In/nState1 @bit 2 <-> ENC Status Channel 1/Status/Set counter done
//     Enc/Inputs/In/nState2 <-> ENC Status Channel 1/Status/Status of input A
//     Enc/Inputs/In/nState2 @bit 1 <-> ENC Status Channel 1/Status/Status of input B
//     Enc/Inputs/In/nState2 @bit 3 <-> ENC Status Channel 1/Status/Status of input gate
//     Enc/Inputs/In/nState4 @bit 1 <-> WcState/InputToggle
//     Enc/Inputs/In/nState4 <-> WcState/WcState
//     Enc/Outputs/Out/nCtrl1 @bit 3 <-> ENC Control Channel 1/Control/Enable latch extern on negative edge
//     Enc/Outputs/Out/nCtrl1 @bit 1 <-> ENC Control Channel 1/Control/Enable latch extern on positive edge
//     Enc/Outputs/Out/nCtrl1 @bit 2 <-> ENC Control Channel 1/Control/Set counter
//     Enc/Outputs/Out/nCtrl2 @bit 2 <-> ENC Control Channel 1/Control/Set counter on latch extern on negative edge
//     Enc/Outputs/Out/nCtrl2 @bit 1 <-> ENC Control Channel 1/Control/Set counter on latch extern on positive edge
//     Enc/Outputs/Out/nCtrl2 <-> ENC Control Channel 1/Control/Set software gate
//     Enc/Outputs/Out/nDataOut1 <-> ENC Control Channel 1/Set counter value
//   (this object) <-> Device 1 (EtherCAT)/Term 5 (EK1200)/Term 6 (EK1122-0080)/DRL02-EK0 (EK1101-0080)/DRL02-E25 (EL5042)
//     Enc/Inputs/In/nComState @bit 1 <-> WcState/InputToggle
//     Enc/Inputs/In/nComState <-> WcState/WcState
//     Enc/Inputs/In/nDataIn1 <-> FB Inputs Channel 2/Position
//     Enc/Inputs/In/nState1 @bit 12 <-> FB Inputs Channel 2/Status/Diag
//     Enc/Inputs/In/nState1 @bit 1 <-> FB Inputs Channel 2/Status/Error
//     Enc/Inputs/In/nState1 @bit 14 <-> FB Inputs Channel 2/Status/Input cycle counter
//     Enc/Inputs/In/nState1 @bit 2 <-> FB Inputs Channel 2/Status/Ready
//     Enc/Inputs/In/nState1 @bit 13 <-> FB Inputs Channel 2/Status/TxPDO State
//     Enc/Inputs/In/nState1 <-> FB Inputs Channel 2/Status/Warning
//   (this object) <-> Device 1 (EtherCAT)/Term 5 (EK1200)/Term 6 (EK1122-0080)/DRL02-EK0 (EK1101-0080)/DRL02-E26 (EL7031)
//     Drive/Inputs/In/nState1 @bit 3 <-> STM Status/Status/Error
//     Drive/Inputs/In/nState1 @bit 5 <-> STM Status/Status/Moving negative
//     Drive/Inputs/In/nState1 @bit 4 <-> STM Status/Status/Moving positive
//     Drive/Inputs/In/nState1 @bit 1 <-> STM Status/Status/Ready
//     Drive/Inputs/In/nState1 <-> STM Status/Status/Ready to enable
//     Drive/Inputs/In/nState1 @bit 6 <-> STM Status/Status/Torque reduced
//     Drive/Inputs/In/nState1 @bit 2 <-> STM Status/Status/Warning
//     Drive/Inputs/In/nState2 @bit 3 <-> STM Status/Status/Digital input 1
//     Drive/Inputs/In/nState2 @bit 4 <-> STM Status/Status/Digital input 2
//     Drive/Inputs/In/nState2 @bit 5 <-> STM Status/Status/Sync error
//     Drive/Inputs/In/nState2 @bit 7 <-> STM Status/Status/TxPDO Toggle
//     Drive/Inputs/In/nState4 @bit 1 <-> WcState/InputToggle
//     Drive/Inputs/In/nState4 <-> WcState/WcState
//     Drive/Outputs/Out/nCtrl1 <-> STM Control/Control/Enable
//     Drive/Outputs/Out/nCtrl1 @bit 2 <-> STM Control/Control/Reduce torque
//     Drive/Outputs/Out/nCtrl1 @bit 1 <-> STM Control/Control/Reset
//     Drive/Outputs/Out/nDataOut2[0] <-> STM Velocity/Velocity
//   (this object) <-> Device 1 (EtherCAT)/Term 5 (EK1200)/Term 6 (EK1122-0080)/DRL02-EK0 (EK1101-0080)/DRL02-E27 (EL7031)
//     Drive/Inputs/In/nState1 @bit 3 <-> STM Status/Status/Error
//     Drive/Inputs/In/nState1 @bit 5 <-> STM Status/Status/Moving negative
//     Drive/Inputs/In/nState1 @bit 4 <-> STM Status/Status/Moving positive
//     Drive/Inputs/In/nState1 @bit 1 <-> STM Status/Status/Ready
//     Drive/Inputs/In/nState1 <-> STM Status/Status/Ready to enable
//     Drive/Inputs/In/nState1 @bit 6 <-> STM Status/Status/Torque reduced
//     Drive/Inputs/In/nState1 @bit 2 <-> STM Status/Status/Warning
//     Drive/Inputs/In/nState2 @bit 3 <-> STM Status/Status/Digital input 1
//     Drive/Inputs/In/nState2 @bit 4 <-> STM Status/Status/Digital input 2
//     Drive/Inputs/In/nState2 @bit 5 <-> STM Status/Status/Sync error
//     Drive/Inputs/In/nState2 @bit 7 <-> STM Status/Status/TxPDO Toggle
//     Drive/Inputs/In/nState4 @bit 1 <-> WcState/InputToggle
//     Drive/Inputs/In/nState4 <-> WcState/WcState
//     Drive/Outputs/Out/nCtrl1 <-> STM Control/Control/Enable
//     Drive/Outputs/Out/nCtrl1 @bit 2 <-> STM Control/Control/Reduce torque
//     Drive/Outputs/Out/nCtrl1 @bit 1 <-> STM Control/Control/Reset
//     Drive/Outputs/Out/nDataOut2[0] <-> STM Velocity/Velocity
//     Enc/Inputs/In/nDataIn1[0] <-> ENC Status compact/Counter value
//     Enc/Inputs/In/nDataIn2[0] <-> ENC Status compact/Latch value
//     Enc/Inputs/In/nState1 @bit 4 <-> ENC Status compact/Status/Counter overflow
//     Enc/Inputs/In/nState1 @bit 3 <-> ENC Status compact/Status/Counter underflow
//     Enc/Inputs/In/nState1 @bit 1 <-> ENC Status compact/Status/Latch extern valid
//     Enc/Inputs/In/nState1 @bit 2 <-> ENC Status compact/Status/Set counter done
//     Enc/Inputs/In/nState2 @bit 4 <-> ENC Status compact/Status/Status of extern latch
//     Enc/Inputs/In/nState2 @bit 5 <-> ENC Status compact/Status/Sync error
//     Enc/Inputs/In/nState2 @bit 7 <-> ENC Status compact/Status/TxPDO Toggle
//     Enc/Inputs/In/nState4 @bit 1 <-> WcState/InputToggle
//     Enc/Inputs/In/nState4 <-> WcState/WcState
//     Enc/Outputs/Out/nCtrl1 @bit 3 <-> ENC Control compact/Control/Enable latch extern on negative edge
//     Enc/Outputs/Out/nCtrl1 @bit 1 <-> ENC Control compact/Control/Enable latch extern on positive edge
//     Enc/Outputs/Out/nCtrl1 @bit 2 <-> ENC Control compact/Control/Set counter
//     Enc/Outputs/Out/nDataOut1[0] <-> ENC Control compact/Set counter value
//   (this object) <-> Device 1 (EtherCAT)/Term 5 (EK1200)/Term 6 (EK1122-0080)/DRL02-EK0 (EK1101-0080)/DRL02-E29 (EL7031)
//     Drive/Inputs/In/nState1 @bit 3 <-> STM Status/Status/Error
//     Drive/Inputs/In/nState1 @bit 5 <-> STM Status/Status/Moving negative
//     Drive/Inputs/In/nState1 @bit 4 <-> STM Status/Status/Moving positive
//     Drive/Inputs/In/nState1 @bit 1 <-> STM Status/Status/Ready
//     Drive/Inputs/In/nState1 <-> STM Status/Status/Ready to enable
//     Drive/Inputs/In/nState1 @bit 6 <-> STM Status/Status/Torque reduced
//     Drive/Inputs/In/nState1 @bit 2 <-> STM Status/Status/Warning
//     Drive/Inputs/In/nState2 @bit 3 <-> STM Status/Status/Digital input 1
//     Drive/Inputs/In/nState2 @bit 4 <-> STM Status/Status/Digital input 2
//     Drive/Inputs/In/nState2 @bit 5 <-> STM Status/Status/Sync error
//     Drive/Inputs/In/nState2 @bit 7 <-> STM Status/Status/TxPDO Toggle
//     Drive/Inputs/In/nState4 @bit 1 <-> WcState/InputToggle
//     Drive/Inputs/In/nState4 <-> WcState/WcState
//     Drive/Outputs/Out/nCtrl1 <-> STM Control/Control/Enable
//     Drive/Outputs/Out/nCtrl1 @bit 2 <-> STM Control/Control/Reduce torque
//     Drive/Outputs/Out/nCtrl1 @bit 1 <-> STM Control/Control/Reset
//     Drive/Outputs/Out/nDataOut2[0] <-> STM Velocity/Velocity
//     Enc/Inputs/In/nDataIn1[0] <-> ENC Status compact/Counter value
//     Enc/Inputs/In/nDataIn2[0] <-> ENC Status compact/Latch value
//     Enc/Inputs/In/nState1 @bit 4 <-> ENC Status compact/Status/Counter overflow
//     Enc/Inputs/In/nState1 @bit 3 <-> ENC Status compact/Status/Counter underflow
//     Enc/Inputs/In/nState1 @bit 1 <-> ENC Status compact/Status/Latch extern valid
//     Enc/Inputs/In/nState1 @bit 2 <-> ENC Status compact/Status/Set counter done
//     Enc/Inputs/In/nState2 @bit 4 <-> ENC Status compact/Status/Status of extern latch
//     Enc/Inputs/In/nState2 @bit 5 <-> ENC Status compact/Status/Sync error
//     Enc/Inputs/In/nState2 @bit 7 <-> ENC Status compact/Status/TxPDO Toggle
//     Enc/Inputs/In/nState4 @bit 1 <-> WcState/InputToggle
//     Enc/Inputs/In/nState4 <-> WcState/WcState
//     Enc/Outputs/Out/nCtrl1 @bit 3 <-> ENC Control compact/Control/Enable latch extern on negative edge
//     Enc/Outputs/Out/nCtrl1 @bit 1 <-> ENC Control compact/Control/Enable latch extern on positive edge
//     Enc/Outputs/Out/nCtrl1 @bit 2 <-> ENC Control compact/Control/Set counter
//     Enc/Outputs/Out/nDataOut1[0] <-> ENC Control compact/Set counter value
//   (this object) <-> Device 1 (EtherCAT)/Term 5 (EK1200)/Term 6 (EK1122-0080)/DRL02-EK0 (EK1101-0080)/DRL02-E30 (EL7031)
//     Drive/Inputs/In/nState1 @bit 3 <-> STM Status/Status/Error
//     Drive/Inputs/In/nState1 @bit 5 <-> STM Status/Status/Moving negative
//     Drive/Inputs/In/nState1 @bit 4 <-> STM Status/Status/Moving positive
//     Drive/Inputs/In/nState1 @bit 1 <-> STM Status/Status/Ready
//     Drive/Inputs/In/nState1 <-> STM Status/Status/Ready to enable
//     Drive/Inputs/In/nState1 @bit 6 <-> STM Status/Status/Torque reduced
//     Drive/Inputs/In/nState1 @bit 2 <-> STM Status/Status/Warning
//     Drive/Inputs/In/nState2 @bit 3 <-> STM Status/Status/Digital input 1
//     Drive/Inputs/In/nState2 @bit 4 <-> STM Status/Status/Digital input 2
//     Drive/Inputs/In/nState2 @bit 5 <-> STM Status/Status/Sync error
//     Drive/Inputs/In/nState2 @bit 7 <-> STM Status/Status/TxPDO Toggle
//     Drive/Inputs/In/nState4 @bit 1 <-> WcState/InputToggle
//     Drive/Inputs/In/nState4 <-> WcState/WcState
//     Drive/Outputs/Out/nCtrl1 <-> STM Control/Control/Enable
//     Drive/Outputs/Out/nCtrl1 @bit 2 <-> STM Control/Control/Reduce torque
//     Drive/Outputs/Out/nCtrl1 @bit 1 <-> STM Control/Control/Reset
//     Drive/Outputs/Out/nDataOut2[0] <-> STM Velocity/Velocity
//     Enc/Inputs/In/nDataIn1[0] <-> ENC Status compact/Counter value
//     Enc/Inputs/In/nDataIn2[0] <-> ENC Status compact/Latch value
//     Enc/Inputs/In/nState1 @bit 4 <-> ENC Status compact/Status/Counter overflow
//     Enc/Inputs/In/nState1 @bit 3 <-> ENC Status compact/Status/Counter underflow
//     Enc/Inputs/In/nState1 @bit 1 <-> ENC Status compact/Status/Latch extern valid
//     Enc/Inputs/In/nState1 @bit 2 <-> ENC Status compact/Status/Set counter done
//     Enc/Inputs/In/nState2 @bit 4 <-> ENC Status compact/Status/Status of extern latch
//     Enc/Inputs/In/nState2 @bit 5 <-> ENC Status compact/Status/Sync error
//     Enc/Inputs/In/nState2 @bit 7 <-> ENC Status compact/Status/TxPDO Toggle
//     Enc/Inputs/In/nState4 @bit 1 <-> WcState/InputToggle
//     Enc/Inputs/In/nState4 <-> WcState/WcState
//     Enc/Outputs/Out/nCtrl1 @bit 3 <-> ENC Control compact/Control/Enable latch extern on negative edge
//     Enc/Outputs/Out/nCtrl1 @bit 1 <-> ENC Control compact/Control/Enable latch extern on positive edge
//     Enc/Outputs/Out/nCtrl1 @bit 2 <-> ENC Control compact/Control/Set counter
//     Enc/Outputs/Out/nDataOut1[0] <-> ENC Control compact/Set counter value
//   (this object) <-> Device 1 (EtherCAT)/Term 5 (EK1200)/Term 6 (EK1122-0080)/DRL02-EK0 (EK1101-0080)/DRL02-E33 (EL7031)
//     Drive/Inputs/In/nState1 @bit 3 <-> STM Status/Status/Error
//     Drive/Inputs/In/nState1 @bit 5 <-> STM Status/Status/Moving negative
//     Drive/Inputs/In/nState1 @bit 4 <-> STM Status/Status/Moving positive
//     Drive/Inputs/In/nState1 @bit 1 <-> STM Status/Status/Ready
//     Drive/Inputs/In/nState1 <-> STM Status/Status/Ready to enable
//     Drive/Inputs/In/nState1 @bit 6 <-> STM Status/Status/Torque reduced
//     Drive/Inputs/In/nState1 @bit 2 <-> STM Status/Status/Warning
//     Drive/Inputs/In/nState2 @bit 3 <-> STM Status/Status/Digital input 1
//     Drive/Inputs/In/nState2 @bit 4 <-> STM Status/Status/Digital input 2
//     Drive/Inputs/In/nState2 @bit 5 <-> STM Status/Status/Sync error
//     Drive/Inputs/In/nState2 @bit 7 <-> STM Status/Status/TxPDO Toggle
//     Drive/Inputs/In/nState4 @bit 1 <-> WcState/InputToggle
//     Drive/Inputs/In/nState4 <-> WcState/WcState
//     Drive/Outputs/Out/nCtrl1 <-> STM Control/Control/Enable
//     Drive/Outputs/Out/nCtrl1 @bit 2 <-> STM Control/Control/Reduce torque
//     Drive/Outputs/Out/nCtrl1 @bit 1 <-> STM Control/Control/Reset
//     Drive/Outputs/Out/nDataOut2[0] <-> STM Velocity/Velocity
//   (this object) <-> Device 1 (EtherCAT)/Term 5 (EK1200)/Term 6 (EK1122-0080)/DRL02-EK0 (EK1101-0080)/DRL02-E31 (EL7031)
//     Drive/Inputs/In/nState1 @bit 3 <-> STM Status/Status/Error
//     Drive/Inputs/In/nState1 @bit 5 <-> STM Status/Status/Moving negative
//     Drive/Inputs/In/nState1 @bit 4 <-> STM Status/Status/Moving positive
//     Drive/Inputs/In/nState1 @bit 1 <-> STM Status/Status/Ready
//     Drive/Inputs/In/nState1 <-> STM Status/Status/Ready to enable
//     Drive/Inputs/In/nState1 @bit 6 <-> STM Status/Status/Torque reduced
//     Drive/Inputs/In/nState1 @bit 2 <-> STM Status/Status/Warning
//     Drive/Inputs/In/nState2 @bit 3 <-> STM Status/Status/Digital input 1
//     Drive/Inputs/In/nState2 @bit 4 <-> STM Status/Status/Digital input 2
//     Drive/Inputs/In/nState2 @bit 5 <-> STM Status/Status/Sync error
//     Drive/Inputs/In/nState2 @bit 7 <-> STM Status/Status/TxPDO Toggle
//     Drive/Inputs/In/nState4 @bit 1 <-> WcState/InputToggle
//     Drive/Inputs/In/nState4 <-> WcState/WcState
//     Drive/Outputs/Out/nCtrl1 <-> STM Control/Control/Enable
//     Drive/Outputs/Out/nCtrl1 @bit 2 <-> STM Control/Control/Reduce torque
//     Drive/Outputs/Out/nCtrl1 @bit 1 <-> STM Control/Control/Reset
//     Drive/Outputs/Out/nDataOut2[0] <-> STM Velocity/Velocity
//   (this object) <-> Device 1 (EtherCAT)/Term 5 (EK1200)/Term 6 (EK1122-0080)/DRL02-EK0 (EK1101-0080)/DRL02-E32 (EL5042)
//     Enc/Inputs/In/nComState @bit 1 <-> WcState/InputToggle
//     Enc/Inputs/In/nComState <-> WcState/WcState
//     Enc/Inputs/In/nDataIn1 <-> FB Inputs Channel 1/Position
//     Enc/Inputs/In/nState1 @bit 12 <-> FB Inputs Channel 1/Status/Diag
//     Enc/Inputs/In/nState1 @bit 1 <-> FB Inputs Channel 1/Status/Error
//     Enc/Inputs/In/nState1 @bit 14 <-> FB Inputs Channel 1/Status/Input cycle counter
//     Enc/Inputs/In/nState1 @bit 2 <-> FB Inputs Channel 1/Status/Ready
//     Enc/Inputs/In/nState1 @bit 13 <-> FB Inputs Channel 1/Status/TxPDO State
//     Enc/Inputs/In/nState1 <-> FB Inputs Channel 1/Status/Warning
//   (this object) <-> Device 1 (EtherCAT)/Term 5 (EK1200)/Term 6 (EK1122-0080)/DRL02-EK0 (EK1101-0080)/DRL02-E28 (EL5042)
//     Enc/Inputs/In/nComState @bit 1 <-> WcState/InputToggle
//     Enc/Inputs/In/nComState <-> WcState/WcState
//     Enc/Inputs/In/nDataIn1 <-> FB Inputs Channel 1/Position
//     Enc/Inputs/In/nState1 @bit 12 <-> FB Inputs Channel 1/Status/Diag
//     Enc/Inputs/In/nState1 @bit 1 <-> FB Inputs Channel 1/Status/Error
//     Enc/Inputs/In/nState1 @bit 14 <-> FB Inputs Channel 1/Status/Input cycle counter
//     Enc/Inputs/In/nState1 @bit 2 <-> FB Inputs Channel 1/Status/Ready
//     Enc/Inputs/In/nState1 @bit 13 <-> FB Inputs Channel 1/Status/TxPDO State
//     Enc/Inputs/In/nState1 <-> FB Inputs Channel 1/Status/Warning
//   Motion Instance <-> Device 1 (EtherCAT)/Term 5 (EK1200)/Term 6 (EK1122-0080)/DRL02-EK0 (EK1101-0080)/DRL02-E1 (EL7031)
//     PlcTask Inputs/Main.stDPXMotor.bLimitBackwardEnable <-> STM Status/Status/Digital input 2
//     PlcTask Inputs/Main.stDPXMotor.bLimitForwardEnable <-> STM Status/Status/Digital input 1
//   Motion Instance <-> Device 1 (EtherCAT)/Term 5 (EK1200)/Term 6 (EK1122-0080)/DRL02-EK0 (EK1101-0080)/DRL02-E3 (EL7031)
//     PlcTask Inputs/Main.stDPYMotor.bLimitBackwardEnable <-> STM Status/Status/Digital input 2
//     PlcTask Inputs/Main.stDPYMotor.bLimitForwardEnable <-> STM Status/Status/Digital input 1
//   Motion Instance <-> Device 1 (EtherCAT)/Term 5 (EK1200)/Term 6 (EK1122-0080)/DRL02-EK0 (EK1101-0080)/DRL02-E4 (EL7031)
//     PlcTask Inputs/Main.stDPZMotor.bLimitBackwardEnable <-> STM Status/Status/Digital input 2
//     PlcTask Inputs/Main.stDPZMotor.bLimitForwardEnable <-> STM Status/Status/Digital input 1
//   Motion Instance <-> NC-Task 1 SAF/Axes/Axis 1 - Diagnostic Paddle X
//     PlcTask Inputs/Main.stDPXMotor.Axis.NcToPlc <-> Outputs/ToPlc
//     PlcTask Outputs/Main.stDPXMotor.Axis.PlcToNc <-> Inputs/FromPlc
//   Motion Instance <-> NC-Task 1 SAF/Axes/Axis 10 - Illumination Y
//     PlcTask Inputs/Main.stILMYMotor.Axis.NcToPlc <-> Outputs/ToPlc
//     PlcTask Outputs/Main.stILMYMotor.Axis.PlcToNc <-> Inputs/FromPlc
//   Motion Instance <-> NC-Task 1 SAF/Axes/Axis 11 - Illumination Z
//     PlcTask Inputs/Main.stILMZMotor.Axis.NcToPlc <-> Outputs/ToPlc
//     PlcTask Outputs/Main.stILMZMotor.Axis.PlcToNc <-> Inputs/FromPlc
//   Motion Instance <-> NC-Task 1 SAF/Axes/Axis 12 - Questar X
//     PlcTask Inputs/Main.stQSTXMotor.Axis.NcToPlc <-> Outputs/ToPlc
//     PlcTask Outputs/Main.stQSTXMotor.Axis.PlcToNc <-> Inputs/FromPlc
//   Motion Instance <-> NC-Task 1 SAF/Axes/Axis 13 - Questar Y
//     PlcTask Inputs/Main.stQSTYMotor.Axis.NcToPlc <-> Outputs/ToPlc
//     PlcTask Outputs/Main.stQSTYMotor.Axis.PlcToNc <-> Inputs/FromPlc
//   Motion Instance <-> NC-Task 1 SAF/Axes/Axis 16 - SDS Injector X
//     PlcTask Inputs/Main.stSDSXMotor.Axis.NcToPlc <-> Outputs/ToPlc
//     PlcTask Outputs/Main.stSDSXMotor.Axis.PlcToNc <-> Inputs/FromPlc
//   Motion Instance <-> NC-Task 1 SAF/Axes/Axis 17 - SDS Injectory Y
//     PlcTask Inputs/Main.stSDSYMotor.Axis.NcToPlc <-> Outputs/ToPlc
//     PlcTask Outputs/Main.stSDSYMotor.Axis.PlcToNc <-> Inputs/FromPlc
//   Motion Instance <-> NC-Task 1 SAF/Axes/Axis 18 - SDS Injector Z
//     PlcTask Inputs/Main.stSDSZMotor.Axis.NcToPlc <-> Outputs/ToPlc
//     PlcTask Outputs/Main.stSDSZMotor.Axis.PlcToNc <-> Inputs/FromPlc
//   Motion Instance <-> NC-Task 1 SAF/Axes/Axis 19 - SDS Rotation Y
//     PlcTask Inputs/Main.stSDSRotMotor.Axis.NcToPlc <-> Outputs/ToPlc
//     PlcTask Outputs/Main.stSDSRotMotor.Axis.PlcToNc <-> Inputs/FromPlc
//   Motion Instance <-> NC-Task 1 SAF/Axes/Axis 2 - Diagnostic Paddle Y
//     PlcTask Inputs/Main.stDPYMotor.Axis.NcToPlc <-> Outputs/ToPlc
//     PlcTask Outputs/Main.stDPYMotor.Axis.PlcToNc <-> Inputs/FromPlc
//   Motion Instance <-> NC-Task 1 SAF/Axes/Axis 20 - SDS Shroud Rotation
//     PlcTask Inputs/Main.stSDSShroudMotor.Axis.NcToPlc <-> Outputs/ToPlc
//     PlcTask Outputs/Main.stSDSShroudMotor.Axis.PlcToNc <-> Inputs/FromPlc
//   Motion Instance <-> NC-Task 1 SAF/Axes/Axis 3 - Diagnostic Paddle Z
//     PlcTask Inputs/Main.stDPZMotor.Axis.NcToPlc <-> Outputs/ToPlc
//     PlcTask Outputs/Main.stDPZMotor.Axis.PlcToNc <-> Inputs/FromPlc
//   Motion Instance <-> NC-Task 1 SAF/Axes/Axis 4 - Objectives X
//     PlcTask Inputs/Main.stOBJXMotor.Axis.NcToPlc <-> Outputs/ToPlc
//     PlcTask Outputs/Main.stOBJXMotor.Axis.PlcToNc <-> Inputs/FromPlc
//   Motion Instance <-> NC-Task 1 SAF/Axes/Axis 5 - Objectives Y
//     PlcTask Inputs/Main.stOBJYMotor.Axis.NcToPlc <-> Outputs/ToPlc
//     PlcTask Outputs/Main.stOBJYMotor.Axis.PlcToNc <-> Inputs/FromPlc
//   Motion Instance <-> NC-Task 1 SAF/Axes/Axis 6 - Objectives Z
//     PlcTask Inputs/Main.stOBJZMotor.Axis.NcToPlc <-> Outputs/ToPlc
//     PlcTask Outputs/Main.stOBJZMotor.Axis.PlcToNc <-> Inputs/FromPlc
//   Motion Instance <-> NC-Task 1 SAF/Axes/Axis 7 - Point Detector Y
//     PlcTask Inputs/Main.stPDYMotor.Axis.NcToPlc <-> Outputs/ToPlc
//     PlcTask Outputs/Main.stPDYMotor.Axis.PlcToNc <-> Inputs/FromPlc
//   Motion Instance <-> NC-Task 1 SAF/Axes/Axis 8 - Point Detector Rotation
//     PlcTask Inputs/Main.stPDRotMotor.Axis.NcToPlc <-> Outputs/ToPlc
//     PlcTask Outputs/Main.stPDRotMotor.Axis.PlcToNc <-> Inputs/FromPlc
//   Motion Instance <-> NC-Task 1 SAF/Axes/Axis 9 - Illumination X
//     PlcTask Inputs/Main.stILMXMotor.Axis.NcToPlc <-> Outputs/ToPlc
//     PlcTask Outputs/Main.stILMXMotor.Axis.PlcToNc <-> Inputs/FromPlc

CONFIGURATION Motion
    RESOURCE PLC ON TwinCAT3
        TASK PlcTask(INTERVAL := T#10ms, PRIORITY := 20);
        PROGRAM PRG_Main WITH PlcTask : PRG_Main;
    END_RESOURCE
END_CONFIGURATION

// ---- DUTs/Assemblies/ENUM_DiagPaddle.TcDUT
{attribute 'qualified_only'}
{attribute 'strict'}
TYPE ENUM_DiagPaddle :
(
	UNKNOWN := 0,
	PARK :=1,
	UP := 2,
	CENTER := 3,
	PINHOLE := 4,
	DIODE := 5,
	YAG1 := 6,
	YAG2 := 7,
	YAG3 := 8,
	KNIFE := 9
);
END_TYPE

// ---- DUTs/Assemblies/ENUM_DPX.TcDUT
{attribute 'qualified_only'}
// EPICS states enum for use in FB_DPX (diagnostic paddle X)
// Remove strict attribute for easier handling
TYPE ENUM_DPX :
(
    UNKNOWN := 0, // UNKNOWN must be in slot 0 or the FB breaks
    PARK := 1,    // The parked position for the diagnostic paddle
    CENTER := 2,  // center positon for the diagnostic paddle. This should be 
	KNIFE	:= 3  // Knife edge position for the diagnostic paddle. Should be the same nominal X positon as the "CENTER"
				  // position, but will use a different set of soft limits to allow scanning of the knife edge.
);
END_TYPE

// ---- DUTs/Assemblies/ENUM_DPY.TcDUT
{attribute 'qualified_only'}
// EPICS states enum for use in FB_DPY (diagnostic paddle Y)
// Remove strict attribute for easier handling
TYPE ENUM_DPY :
(
    UNKNOWN := 0,	// UNKNOWN must be in slot 0 or the FB breaks
    PARK := 1,		// The parked position for the diagnostic paddle
    CENTER := 2,	// center positon for the diagnostic paddle. This should be 
	PINHOLE	:= 3,   // Pinhole position for WFS
	DIODE :=4,		// Diode position
	YAG1 := 5,		// Yag 1 position
	YAG2 := 6,		// Yag 2 position
	YAG3 := 7,		// Yag 3 position
	KNIFE := 8 	    // Knife edge position for the diagnostic paddle. Should be the same nominal X positon as the "CENTER"
				    // position, but will use a different set of soft limits to allow scanning of the knife edge.
);
END_TYPE

// ---- DUTs/Assemblies/E_DPaddle_States.TcDUT
{attribute 'qualified_only'}
{attribute 'strict'}
TYPE E_DPaddle_States :
(
	parked := 0,
	diode,
	L1,
	L2,
	L3,
	L4,
	R1,
	R2,
	R3,
	R4
);
END_TYPE

// ---- GVLs/GVL.TcGVL
{attribute 'qualified_only'}
VAR_GLOBAL	
	xOverride		:	BOOL := FALSE; // Global override of motion safety settings.
END_VAR

// ---- GVLs/GVL_DiagnosticPaddle.TcGVL
VAR_GLOBAL
	

							
	// Define axis states for each axis. These are fed to a FB_PositionState manager for each axis
	// X axis position states
	stDPXPosPark : DUT_PositionState :=		(sName:= 'PARK',
										 	fPosition := 5.0,
										 	fDelta:=1.0,
									     	fVelocity:=5.0,
    									 	fAccel:=1.0, 
											fDecel:=1.0,
    									 	bMoveOk:=FALSE,
    									 	bLocked:=TRUE,
    									 	bValid:=TRUE);
	stDPXPosCenter : DUT_PositionState :=	(sName:= 'CENTER',
										 	fPosition := 10.0,
										 	fDelta:=1.0,
									     	fVelocity:=5.0,
    									 	fAccel:=1.0, 
										 	fDecel:=1.0,
    										bMoveOk:=FALSE,
    									 	bLocked:=TRUE,
    									 	bValid:=TRUE);
	stDPXPosKnife : DUT_PositionState :=	(sName:= 'KNIFE',
										 	fPosition := 15.0,
										 	fDelta:=1.0,
									     	fVelocity:=5.0,
    									 	fAccel:=1.0, 
										 	fDecel:=1.0,
    										bMoveOk:=FALSE,
    									 	bLocked:=TRUE,
    									 	bValid:=TRUE);
											


	// Y axis position states
	stDPYPosPark : DUT_PositionState :=		(sName:= 'PARK',
										 	fPosition := 5.0,
										 	fDelta:=1.0,
									     	fVelocity:=5.0,
    									 	fAccel:=1.0, 
											fDecel:=1.0,
    									 	bMoveOk:=FALSE,
    									 	bLocked:=TRUE,
    									 	bValid:=TRUE);
	stDPYPosCenter : DUT_PositionState :=	(sName:= 'CENTER',
										 	fPosition := 10.0,
										 	fDelta:=1.0,
									     	fVelocity:=5.0,
    									 	fAccel:=1.0, 
										 	fDecel:=1.0,
    										bMoveOk:=FALSE,
    									 	bLocked:=TRUE,
    									 	bValid:=TRUE);
	stDPYPosDiode : DUT_PositionState :=	(sName:= 'DIODE',
										 	fPosition := 15.0,
										 	fDelta:=1.0,
									     	fVelocity:=5.0,
    									 	fAccel:=1.0, 
											fDecel:=1.0,
    									 	bMoveOk:=FALSE,
    									 	bLocked:=TRUE,
    									 	bValid:=TRUE);
	stDPYPosPinhole : DUT_PositionState :=	(sName:= 'PINHOLE',
										 	fPosition := 20.0,
										 	fDelta:=1.0,
									     	fVelocity:=5.0,
    									 	fAccel:=1.0, 
										 	fDecel:=1.0,
    										bMoveOk:=FALSE,
    									 	bLocked:=TRUE,
    									 	bValid:=TRUE);
	stDPYPosYAG1 : DUT_PositionState :=		(sName:= 'YAG1',
										 	fPosition := 25.0,
										 	fDelta:=1.0,
									     	fVelocity:=5.0,
    									 	fAccel:=1.0, 
										 	fDecel:=1.0,
    										bMoveOk:=FALSE,
    									 	bLocked:=TRUE,
    									 	bValid:=TRUE);
	stDPYPosYAG2 : DUT_PositionState :=		(sName:= 'YAG2',
										 	fPosition := 30.0,
										 	fDelta:=1.0,
									     	fVelocity:=5.0,
    									 	fAccel:=1.0, 
										 	fDecel:=1.0,
    										bMoveOk:=FALSE,
    									 	bLocked:=TRUE,
    									 	bValid:=TRUE);
	stDPYPosYAG3 : DUT_PositionState :=		(sName:= 'YAG3',
										 	fPosition := 35.0,
										 	fDelta:=1.0,
									     	fVelocity:=5.0,
    									 	fAccel:=1.0, 
										 	fDecel:=1.0,
    										bMoveOk:=FALSE,
    									 	bLocked:=TRUE,
    									 	bValid:=TRUE);
	stDPYPosKnife : DUT_PositionState :=	(sName:= 'KNIFE',
										 	fPosition := 40.0,
										 	fDelta:=1.0,
									     	fVelocity:=5.0,
    									 	fAccel:=1.0, 
										 	fDecel:=1.0,
    										bMoveOk:=FALSE,
    									 	bLocked:=TRUE,
    									 	bValid:=TRUE);
											
	// Z axis position states						
	stDPZPosPark : DUT_PositionState :=		(sName:= 'PARK',
										 	fPosition := 5.0,
										 	fDelta:=1.0,
									     	fVelocity:=5.0,
    									 	fAccel:=1.0, 
											fDecel:=1.0,
    									 	bMoveOk:=FALSE,
    									 	bLocked:=TRUE,
    									 	bValid:=TRUE);
	stDPZPosCenter : DUT_PositionState :=	(sName:= 'CENTER',
										 	fPosition := 10.0,
										 	fDelta:=1.0,
									     	fVelocity:=5.0,
    									 	fAccel:=1.0, 
										 	fDecel:=1.0,
    										bMoveOk:=FALSE,
    									 	bLocked:=TRUE,
    									 	bValid:=TRUE);
					
	stDPPark 	: ST_BFSAssemblyState := (iState:=1, bDiscovered:=FALSE, iParent:=0);
	stDPUp	 	: ST_BFSAssemblyState := (iState:=2, bDiscovered:=FALSE, iParent:=0);	
	stDPCenter 	: ST_BFSAssemblyState := (iState:=3, bDiscovered:=FALSE, iParent:=0);
	stDPPinhole : ST_BFSAssemblyState := (iState:=4, bDiscovered:=FALSE, iParent:=0);	
	stDPDiode 	: ST_BFSAssemblyState := (iState:=5, bDiscovered:=FALSE, iParent:=0);	
	stDPYag1 	: ST_BFSAssemblyState := (iState:=6, bDiscovered:=FALSE, iParent:=0);	
	stDPYag2 	: ST_BFSAssemblyState := (iState:=7, bDiscovered:=FALSE, iParent:=0);	
	stDPYag3 	: ST_BFSAssemblyState := (iState:=8, bDiscovered:=FALSE, iParent:=0);	
	stDPKnife 	: ST_BFSAssemblyState := (iState:=9, bDiscovered:=FALSE, iParent:=0);	

	arrDPStates : ARRAY [1..9] OF ST_BFSAssemblyState := [stDPPark, stDPUp, stDPCenter, stDPPinhole, stDPDiode,
														  stDPYag1, stDPYag2, stDPYag3, stDPKnife];
	
END_VAR

// ---- GVLs/GVL_Illumination.TcGVL
//{attribute 'qualified_only'}
VAR_GLOBAL
	
	


							
	// Define axis states for each axis. These are fed to a FB_PositionState manager for each axis
	// X axis position states
	stILMXPosPark : DUT_PositionState :=   (sName:= 'PARK',
										 	fPosition := 0.0,
										 	fDelta:=1.0,
									     	fVelocity:=5.0,
    									 	fAccel:=1.0, 
											fDecel:=1.0,
    									 	bMoveOk:=FALSE,
    									 	bLocked:=TRUE,
    									 	bValid:=TRUE);

	// Y axis position states
	stILMYPosPark : DUT_PositionState :=   (sName:= 'PARK',
										 	fPosition := 0.0,
										 	fDelta:=1.0,
									     	fVelocity:=5.0,
    									 	fAccel:=1.0, 
											fDecel:=1.0,
    									 	bMoveOk:=FALSE,
    									 	bLocked:=TRUE,
    									 	bValid:=TRUE);
											
	// Z axis position states						
	stILMZPosPark : DUT_PositionState :=   (sName:= 'PARK',
										 	fPosition := 0.0,
										 	fDelta:=1.0,
									     	fVelocity:=5.0,
    									 	fAccel:=1.0, 
											fDecel:=1.0,
    									 	bMoveOk:=FALSE,
    									 	bLocked:=TRUE,
    									 	bValid:=TRUE);
	
	fbILMXStage : FB_MotionStage;
	fbILMYStage : FB_MotionStage;
	fbILMZStage : FB_MotionStage;
END_VAR

// ---- GVLs/GVL_Objectives.TcGVL
{attribute 'qualified_only'}
VAR_GLOBAL
	// Motor axes
	stOBJXMotor : DUT_MotionStage;
	stOBJYMotor : DUT_MotionStage;
	stOBJZMotor : DUT_MotionStage;
							
	// Define axis states for each axis. These are fed to a FB_PositionState manager for each axis
	// X axis position states
	stOBJXPosPark : DUT_PositionState :=		(sName:= 'PARK',
										 	fPosition := 0.0,
										 	fDelta:=1.0,
									     	fVelocity:=5.0,
    									 	fAccel:=1.0, 
											fDecel:=1.0,
    									 	bMoveOk:=FALSE,
    									 	bLocked:=TRUE,
    									 	bValid:=TRUE);

	// Y axis position states
	stOBJYPosPark : DUT_PositionState :=		(sName:= 'PARK',
										 	fPosition := -50.0,
										 	fDelta:=1.0,
									     	fVelocity:=5.0,
    									 	fAccel:=1.0, 
											fDecel:=1.0,
    									 	bMoveOk:=FALSE,
    									 	bLocked:=TRUE,
    									 	bValid:=TRUE);
											
	// Z axis position states						
	stOBJZPosPark : DUT_PositionState :=		(sName:= 'PARK',
										 	fPosition := -25.0,
										 	fDelta:=1.0,
									     	fVelocity:=5.0,
    									 	fAccel:=1.0, 
											fDecel:=1.0,
    									 	bMoveOk:=FALSE,
    									 	bLocked:=TRUE,
    									 	bValid:=TRUE);
END_VAR

// ---- GVLs/GVL_PointDetector.TcGVL
{attribute 'qualified_only'}
VAR_GLOBAL
		// Motor axes

							
	// Define axis states for each axis. These are fed to a FB_PositionState manager for each axis
	// Rotation axis position states
	stPDRotPosPark : DUT_PositionState :=		(sName:= 'PARK',
										 	fPosition := 10.0,
										 	fDelta:=1.0,
									     	fVelocity:=5.0,
    									 	fAccel:=1.0, 
											fDecel:=1.0,
    									 	bMoveOk:=FALSE,
    									 	bLocked:=TRUE,
    									 	bValid:=TRUE);

	// Y axis position states
	stPDYPosPark : DUT_PositionState :=		(sName:= 'PARK',
										 	fPosition := 21.0,
										 	fDelta:=1.0,
									     	fVelocity:=5.0,
    									 	fAccel:=1.0, 
											fDecel:=1.0,
    									 	bMoveOk:=FALSE,
    									 	bLocked:=TRUE,
    									 	bValid:=TRUE);
											
END_VAR

// ---- GVLs/GVL_Questar.TcGVL
{attribute 'qualified_only'}
VAR_GLOBAL
		// Motor axes
	stQSTXMotor : DUT_MotionStage;
	stQSTYMotor : DUT_MotionStage;
							
	// Define axis states for each axis. These are fed to a FB_PositionState manager for each axis
	// X axis position states
	stQSTXPosPark : DUT_PositionState :=		(sName:= 'PARK',
										 	fPosition := 0.0,
										 	fDelta:=1.0,
									     	fVelocity:=5.0,
    									 	fAccel:=1.0, 
											fDecel:=1.0,
    									 	bMoveOk:=FALSE,
    									 	bLocked:=TRUE,
    									 	bValid:=TRUE);

	// Y axis position states
	stQSTYPosPark : DUT_PositionState :=		(sName:= 'PARK',
										 	fPosition := 0.0,
										 	fDelta:=1.0,
									     	fVelocity:=5.0,
    									 	fAccel:=1.0, 
											fDecel:=1.0,
    									 	bMoveOk:=FALSE,
    									 	bLocked:=TRUE,
    									 	bValid:=TRUE);
										
END_VAR

// ---- GVLs/GVL_SampleDelivery.TcGVL
{attribute 'qualified_only'}
VAR_GLOBAL
		// Motor axes
	stSDSXMotor : DUT_MotionStage;
	stSDSYMotor : DUT_MotionStage;
	stSDSZMotor : DUT_MotionStage;
	stSDSRotMotor : DUT_MotionStage;
	stSDSShroudMotor : DUT_MotionStage;
							
	// Define axis states for each axis. These are fed to a FB_PositionState manager for each axis
	// X axis position states
	stSDSXPosPark : DUT_PositionState :=		(sName:= 'PARK',
										 	fPosition := 5.0,
										 	fDelta:=1.0,
									     	fVelocity:=5.0,
    									 	fAccel:=1.0, 
											fDecel:=1.0,
    									 	bMoveOk:=FALSE,
    									 	bLocked:=TRUE,
    									 	bValid:=TRUE);

	// Y axis position states
	stSDSYPosPark : DUT_PositionState :=		(sName:= 'PARK',
										 	fPosition := 5.0,
										 	fDelta:=1.0,
									     	fVelocity:=5.0,
    									 	fAccel:=1.0, 
											fDecel:=1.0,
    									 	bMoveOk:=FALSE,
    									 	bLocked:=TRUE,
    									 	bValid:=TRUE);
											
	// Z axis position states						
	stSDSZPosPark : DUT_PositionState :=		(sName:= 'PARK',
										 	fPosition := 5.0,
										 	fDelta:=1.0,
									     	fVelocity:=5.0,
    									 	fAccel:=1.0, 
											fDecel:=1.0,
    									 	bMoveOk:=FALSE,
    									 	bLocked:=TRUE,
    									 	bValid:=TRUE);
	// Rotation axis position states						
	stSDSRotPosPark : DUT_PositionState :=		(sName:= 'PARK',
										 		 fPosition := 5.0,
										 	fDelta:=1.0,
									     	fVelocity:=5.0,
    									 	fAccel:=1.0, 
											fDecel:=1.0,
    									 	bMoveOk:=FALSE,
    									 	bLocked:=TRUE,
    									 	bValid:=TRUE);
	// Shroud axis position states						
	stSDSShroudPosPark : DUT_PositionState :=		(sName:= 'PARK',
										 			fPosition := 5.0,
										 	fDelta:=1.0,
									     	fVelocity:=5.0,
    									 	fAccel:=1.0, 
											fDecel:=1.0,
    									 	bMoveOk:=FALSE,
    									 	bLocked:=TRUE,
    									 	bValid:=TRUE);
END_VAR

// ---- GVLs/Main.TcGVL
//{attribute 'qualified_only'}
VAR_GLOBAL

	// Motor axes
    {attribute 'pytmc' := 'pv: CRIX:DPL:MMS:X'}
    {attribute 'TcLinkTo' := '.bLimitForwardEnable  := TIID^Device 1 (EtherCAT)^Term 5 (EK1200)^Term 6 (EK1122-0080)^DRL02-EK0 (EK1101-0080)^DRL02-E1 (EL7031)^STM Status^Status^Digital input 1;
                              .bLimitBackwardEnable := TIID^Device 1 (EtherCAT)^Term 5 (EK1200)^Term 6 (EK1122-0080)^DRL02-EK0 (EK1101-0080)^DRL02-E1 (EL7031)^STM Status^Status^Digital input 2'}
	stDPXMotor : DUT_MotionStage;
	
	{attribute 'pytmc' := 'pv: CRIX:DPL:MMS:Y'}
    {attribute 'TcLinkTo' := '.bLimitForwardEnable  := TIID^Device 1 (EtherCAT)^Term 5 (EK1200)^Term 6 (EK1122-0080)^DRL02-EK0 (EK1101-0080)^DRL02-E3 (EL7031)^STM Status^Status^Digital input 1;
                              .bLimitBackwardEnable := TIID^Device 1 (EtherCAT)^Term 5 (EK1200)^Term 6 (EK1122-0080)^DRL02-EK0 (EK1101-0080)^DRL02-E3 (EL7031)^STM Status^Status^Digital input 2'}
	stDPYMotor : DUT_MotionStage;
	
	{attribute 'pytmc' := 'pv: CRIX:DPL:MMS:Z'}
    {attribute 'TcLinkTo' := '.bLimitForwardEnable  := TIID^Device 1 (EtherCAT)^Term 5 (EK1200)^Term 6 (EK1122-0080)^DRL02-EK0 (EK1101-0080)^DRL02-E4 (EL7031)^STM Status^Status^Digital input 1;
                              .bLimitBackwardEnable := TIID^Device 1 (EtherCAT)^Term 5 (EK1200)^Term 6 (EK1122-0080)^DRL02-EK0 (EK1101-0080)^DRL02-E4 (EL7031)^STM Status^Status^Digital input 2'}
	stDPZMotor : DUT_MotionStage;
	
	stILMXMotor : DUT_MotionStage;
	stILMYMotor : DUT_MotionStage;
	stILMZMotor : DUT_MotionStage;
	
	stOBJXMotor : DUT_MotionStage;
	stOBJYMotor : DUT_MotionStage;
	stOBJZMotor : DUT_MotionStage;
	
	stPDRotMotor : DUT_MotionStage;
	stPDYMotor : DUT_MotionStage;
	
	stQSTXMotor : DUT_MotionStage;
	stQSTYMotor : DUT_MotionStage;
	
	stSDSXMotor : DUT_MotionStage;
	stSDSYMotor : DUT_MotionStage;
	stSDSZMotor : DUT_MotionStage;
	stSDSRotMotor : DUT_MotionStage;
	stSDSShroudMotor : DUT_MotionStage;
	
	
END_VAR

// ---- POUs/PRG_Main.TcPOU
PROGRAM PRG_Main
VAR
	//stTestMotor1	:	DUT_SimMotor;
	//fbTestMotor		:	FB_SIM_MOTOR;
	bInit			:	BOOL := FALSE;
	DPState : INT;
	arrStates : ARRAY [1..9] OF ENUM_DiagPaddle;
	bDPaddleOK : BOOL;
	
END_VAR

IF NOT bInit THEN
	bInit := TRUE;
END_IF

// Add interlock logic to this later
bDPaddleOK := TRUE;
//PRG_DiagnosticPaddle(xMoveOK:=bDPaddleOK);

//PRG_QueueTest();

//PRG_Test_AdjacentStates();	

//PRG_BFS();							

PRG_DiagnosticPaddleMotors();

END_PROGRAM

// ---- POUs/Assemblies/PRG_DiagnosticPaddleMotors.TcPOU
PROGRAM PRG_DiagnosticPaddleMotors
VAR
    fbDPX_Motor : FB_MotionStage;
    fbDPY_Motor : FB_MotionStage;
    fbDPZ_Motor : FB_MotionStage;
END_VAR

fbDPX_Motor(stMotionStage:=Main.stDPXMotor);

fbDPY_Motor(stMotionStage:=Main.stDPYMotor);

fbDPZ_Motor(stMotionStage:=Main.stDPZMotor);

END_PROGRAM

// ---- POUs/Assemblies/FB_DPX.TcPOU
FUNCTION_BLOCK FB_DPX

VAR_IN_OUT
    // Motor to apply states to
    stMotionStage: DUT_MotionStage;
    // Information about the park position
    stPark: DUT_PositionState;
    // Information about the center parameter
    stCenter: DUT_PositionState;
	// Information about the knife edge parameter
	stKnife: DUT_PositionState;
END_VAR
VAR_INPUT
    // If TRUE, the motor will be moved when enumSet is changed
    bEnable: BOOL;
    // When changed, sets the destination and starts a move
    {attribute 'pytmc' := '
        pv: SET
        io: io
    '}
    enumSet: ENUM_DPX;
	bOverride: BOOL; // Override for state locking. If TRUE, do not lock states.
END_VAR
VAR_OUTPUT
    // If TRUE, we are in an error state
    bError: BOOL; // NOTE: do not pragma these, already has pragma in manager
    // Error code
    nErrorId: UDINT;
    // Message associated with bError = TRUE
    sErrorMessage: STRING;
    // If TRUE, we are currently moving between states
    bBusy: BOOL;
    // If TRUE, we asked for a move between states, it completed successfully, and there is no ongoing move
    bDone: BOOL;
    // The current state readback
    {attribute 'pytmc' := '
        pv: GET
        io: i
    '}
    enumGet: ENUM_DPX; // NOTE: Please copy this pragma exactly on your enumGet
END_VAR
VAR
    bInit: BOOL;
    arrStates: ARRAY[1..15] OF DUT_PositionState;

    {attribute 'pytmc' := '
        pv:
        io: io
    '}
    fbStateManager: FB_PositionStateManager; // NOTE: Please copy this pragma exactly to pick up the standard PVs
    fbLockPark: 	FB_PositionStateLock;
    fbLockCenter: 	FB_PositionStateLock;
	fbLockKnife: 	FB_PositionStateLock;
END_VAR

// Fist cycle setup
IF NOT bInit THEN
    stPark.sName := 'PARK';
    stCenter.sName := 'CENTER';
	stKnife.sName := 'KNIFE';
    bInit := TRUE;
END_IF

// If any of these have bLocked = TRUE, do not allow user to change them
IF NOT bOverride THEN
	fbLockPark(stPositionState:=stPark);
	fbLockCenter(stPositionState:=stCenter);
	fbLockKnife(stPositionState:=stKnife);
END_IF

// Stuff values into the 15 element array for the manager
arrStates[1] := stPark;
arrStates[2] := stCenter;
arrStates[3] := stKnife;

// Call the function block every cycle
fbStateManager(
    stMotionStage := stMotionStage,
    arrStates := arrStates,
    setState := enumSet,
    bEnable := bEnable,
    bError => bError,
    nErrorId => nErrorId,
    sErrorMessage => sErrorMessage,
    bBusy => bBusy,
    bDone => bDone,
    getState => enumGet); // Cannot do this assignment if enumGet has attribute strict

END_FUNCTION_BLOCK

// ---- POUs/Assemblies/PRG_Cryopumps.TcPOU
PROGRAM PRG_Cryopumps
VAR
    // Motor axes
	stCP1Motor : DUT_MotionStage;
	stCP2Motor : DUT_MotionStage;
							
	// Define axis states for each axis. These are fed to a FB_PositionState manager for each axis
	// Rotation axis position states
	stCP1PosPark : DUT_PositionState :=		(sName:= 'PARK',
										 	fPosition := 0.0,
										 	fDelta:=1.0,
									     	fVelocity:=5.0,
    									 	fAccel:=1.0, 
											fDecel:=1.0,
    									 	bMoveOk:=FALSE,
    									 	bLocked:=TRUE,
    									 	bValid:=TRUE);

	// Y axis position states
	stCP2PosPark : DUT_PositionState :=		(sName:= 'PARK',
										 	fPosition := 0.0,
										 	fDelta:=1.0,
									     	fVelocity:=5.0,
    									 	fAccel:=1.0, 
											fDecel:=1.0,
    									 	bMoveOk:=FALSE,
    									 	bLocked:=TRUE,
    									 	bValid:=TRUE);
END_VAR

END_PROGRAM

// ---- POUs/Assemblies/PRG_DiagnosticPaddle.TcPOU
PROGRAM PRG_DiagnosticPaddle
(*	Program for the ChemRIXS diagnostic paddle. This program sets up a series of PositionStateManagers to implement
	the necessary logic to protect the assembly from running into the recirculation system tube and catcher. *)
	
	// TODO: Setup position state locks?
VAR_INPUT
	xMoveOK : BOOL := FALSE; // External interlock. Applied to bEnable of all PositionStateManagers.
END_VAR
VAR
	bInit : BOOL := FALSE; // Initialization variable
	iCounter : UDINT; // loop counter
	
	// Setup Assembly manager to set bMoveOK for appropriate states
	fbDPAssemblyManager : FB_AssemblyPositionStatemanager;
	
	// Array of axes for protection FB
	arrDPAxes : ARRAY [1..3] OF DUT_MotionStage := [stDPXMotor, stDPYMotor, stDPZMotor];
	
	//  Setup diagnostic paddle adjacency matrix
	arrDPTransitions : ARRAY [0..9, 1..9] OF BOOL := 	
    //Park  Up     Center Pinh.  Diode  Yag1   Yag2   Yag3   Knife
	[FALSE, FALSE, FALSE, FALSE, FALSE, FALSE, FALSE, FALSE, FALSE, // Unknown (This should always be included)
	 TRUE,  TRUE,  FALSE, FALSE, FALSE, FALSE, FALSE, FALSE, FALSE, // Park
	 TRUE,  TRUE,  TRUE,  FALSE, FALSE, FALSE, FALSE, FALSE, FALSE, // Up
	 TRUE,  TRUE,  TRUE,  TRUE,  TRUE,  TRUE,  TRUE,  TRUE,  TRUE,  // Center
	 FALSE, FALSE, TRUE,  TRUE,  TRUE,  TRUE,  TRUE,  TRUE,  TRUE,  // Pinhole
	 FALSE, FALSE, TRUE,  TRUE,  TRUE,  TRUE,  TRUE,  TRUE,  TRUE,  // Diode
	 FALSE, FALSE, TRUE,  TRUE,  TRUE,  TRUE,  TRUE,  TRUE,  TRUE,  // Yag1
	 FALSE, FALSE, TRUE,  TRUE,  TRUE,  TRUE,  TRUE,  TRUE,  TRUE,  // Yag2
	 FALSE, FALSE, TRUE,  TRUE,  TRUE,  TRUE,  TRUE,  TRUE,  TRUE,  // Yag3
	 FALSE, FALSE, TRUE,  TRUE,  TRUE,  TRUE,  TRUE,  TRUE,  TRUE]; // Knife	
	 
	// Setup diagnostic paddle output matrix
	arrDPOutputs		: ARRAY [1..9, 1..3] OF DUT_PositionState :=
	//X axis		    Y axis			    Z axis		         Assembly state
	[stDPXPosPark,		stDPYPosPark,		stDPZPosPark,	  // Park
	 stDPXPosPark, 		stDPYPosCenter,		stDPZPosPark, 	  // Up
	 stDPXPosCenter, 	stDPYPosCenter,		stDPZPosCenter,   // Center
	 stDPXPosCenter, 	stDPYPosPinhole,	stDPZPosCenter,   // Pinhole
	 stDPXPosCenter,	stDPYPosDiode,		stDPZPosCenter,   // Diode
	 stDPXPosCenter,	stDPYPosYag1,		stDPZPosCenter,   // Yag1
	 stDPXPosCenter,	stDPYPosYag2,		stDPZPosCenter,   // Yag2
	 stDPXPosCenter,	stDPYPosYag3,		stDPZPosCenter,   // Yag3
	 stDPXPosCenter,	stDPYPosKnife,		stDPZPosCenter];  // Knife
	
	// TODO: Figure out a way to make this more useful, or remove it. 
	arrDPStates			: ARRAY[0..9] OF STRING := ['UNKNOWN', 'PARK', 'UP', 'CENTER', 
													'PINHOLE', 'DIODE', 'YAG1', 'YAG2', 
													'YAG3',	'KNIFE'];
					
	// Array of position states for PositionStateManagers (initialize later)
	arrDPXStates : ARRAY [1..15] OF DUT_PositionState;
	arrDPYStates : ARRAY [1..15] OF DUT_PositionState;																  
	arrDPZStates : ARRAY [1..15] OF DUT_PositionState;
									
	// Setup PositionStateManagers and set variables for each axis		
	// X Axis			
	// When changed, sets the destination and starts a move
    {attribute 'pytmc' := '
        pv: SET
        io: io
    '}
    enumDPXSet: ENUM_DPX; // NOTE: Please copy this pragma exactly on your enumSet			
	{attribute 'pytmc' := '
        pv:
       	io: io
    '}
    fbXStateManager: FB_PositionStateManager;
	
	// Y axis
	// When changed, sets the destination and starts a move
    {attribute 'pytmc' := '
        pv: SET
        io: io
    '}
    enumDPYSet: ENUM_DPY; // NOTE: Please copy this pragma exactly on your enumSet	
	{attribute 'pytmc' := '
        pv:
        io: io
    '}
    fbYStateManager: FB_PositionStateManager;
	
	// Z axis
	// When changed, sets the destination and starts a move
    {attribute 'pytmc' := '
        pv: SET
        io: io
    '}
    enumDPZSet: ENUM_DPZ; // NOTE: Please copy this pragma exactly on your enumSet	
	{attribute 'pytmc' := '
        pv:
        io: io
    '}
    fbZStateManager: FB_PositionStateManager;
	
	arrPosLocks : ARRAY [1..13] OF FB_PositionStateLock;
	
END_VAR
VAR_OUTPUT
	// Setup PositionStateManager Outputs
	// X Axis
	// If TRUE, we are in an error state
    bDPXError: BOOL; // NOTE: do not pragma these, already has pragma in manager
    // Error code
    nDPXErrorId: UDINT;
    // Message associated with bError = TRUE
    sDPXErrorMessage: STRING;
    // If TRUE, we are currently moving between states
    bDPXBusy: BOOL;
    // If TRUE, we asked for a move between states, it completed successfully, and there is no ongoing move
    bDPXDone: BOOL;
    // The current state readback
    {attribute 'pytmc' := '
        pv: GET
        io: i
    '}
    enumDPXGet: ENUM_DPX; // NOTE: Please copy this pragma exactly on your enumGet
	
	// Y Axis
	// If TRUE, we are in an error state
    bDPYError: BOOL; // NOTE: do not pragma these, already has pragma in manager
    // Error code
    nDPYErrorId: UDINT;
    // Message associated with bError = TRUE
    sDPYErrorMessage: STRING;
    // If TRUE, we are currently moving between states
    bDPYBusy: BOOL;
    // If TRUE, we asked for a move between states, it completed successfully, and there is no ongoing move
    bDPYDone: BOOL;
    // The current state readback
    {attribute 'pytmc' := '
        pv: GET
        io: i
    '}
    enumDPYGet: ENUM_DPY; // NOTE: Please copy this pragma exactly on your enumGet
		
	// Z Axis
	// If TRUE, we are in an error state
    bDPZError: BOOL; // NOTE: do not pragma these, already has pragma in manager
    // Error code
    nDPZErrorId: UDINT;
    // Message associated with bError = TRUE
    sDPZErrorMessage: STRING;
    // If TRUE, we are currently moving between states
    bDPZBusy: BOOL;
    // If TRUE, we asked for a move between states, it completed successfully, and there is no ongoing move
    bDPZDone: BOOL;
    // The current state readback
    {attribute 'pytmc' := '
        pv: GET
        io: i
    '}
    enumDPZGet: ENUM_DPZ; // NOTE: Please copy this pragma exactly on your enumGet
END_VAR

IF NOT bInit THEN
	// Init X axis array
	arrDPXStates[1] := stDPXPosPark;
	arrDPXStates[2] := stDPXPosCenter;
	arrDPXStates[3] := stDPXPosKnife;
	// Init Y axis array
	arrDPYStates[1] := stDPYPosPark;
	arrDPYStates[2] := stDPYPosCenter;
	arrDPYStates[3] := stDPYPosPinhole;
	arrDPYStates[4] := stDPYPosDiode;
	arrDPYStates[5] := stDPYPosYag1;
	arrDPYStates[6] := stDPYPosYag2;
	arrDPYStates[7] := stDPYPosYag3;
	arrDPYStates[8] := stDPYPosKnife;
	// Init Z axis array
	arrDPZStates[1] := stDPZPosPark;
	arrDPZStates[2] := stDPZPosCenter;
	
	
	bInit := TRUE;
END_IF

// Manage the logic between the Diagnostic Paddle axes
fbDPAssemblyManager(arrOutputs:=arrDPOutputs,
					arrTransitions:=arrDPTransitions,
					arrAxes:=arrDPAxes,
					arrAssemblyStates:=arrDPStates);
					
// Update positions based on motion requests
fbXStateManager(
    stMotionStage := stDPXMotor,
    arrStates := arrDPXStates,
    setState := enumDPXSet,
    bEnable := xMoveOK,
    bError => bDPXError,
    nErrorId => nDPXErrorId,
    sErrorMessage => sDPXErrorMessage,
    bBusy => bDPXBusy,
    bDone => bDPXDone,
    getState => enumDPXGet); 
	
fbYStateManager(
    stMotionStage := stDPYMotor,
    arrStates := arrDPYStates,
    setState := enumDPYSet,
    bEnable := xMoveOK,
    bError => bDPYError,
    nErrorId => nDPYErrorId,
    sErrorMessage => sDPYErrorMessage,
    bBusy => bDPYBusy,
    bDone => bDPYDone,
    getState => enumDPYGet); 
	
fbZStateManager(
    stMotionStage := stDPZMotor,
    arrStates := arrDPZStates,
    setState := enumDPZSet,
    bEnable := xMoveOK,
    bError => bDPZError,
    nErrorId => nDPZErrorId,
    sErrorMessage => sDPZErrorMessage,
    bBusy => bDPZBusy,
    bDone => bDPZDone,
    getState => enumDPZGet);

END_PROGRAM

// ---- POUs/EPS/FB_AssemblyPositionStateManager.TcPOU
FUNCTION_BLOCK FB_AssemblyPositionStateManager
(*
    Handles EPICS moves between multiple states for multiple axes.
    See FB_XXXX for an example.
*)
VAR_IN_OUT

	// Array of bMoveEnables to, well, enable based on the assembly state.
    arrOutputs: ARRAY [*, *] OF DUT_PositionState;
	// Array of allowed position state transitions. This is the adjacency matrix
	arrTransitions : ARRAY [*, *] OF BOOL;
	// Array of all axes in the assembly
	arrAxes : ARRAY [*] OF DUT_MotionStage;
	// Array of all assembly states
	arrAssemblyStates : ARRAY [*] OF STRING;
END_VAR
VAR	
	nAssemblyStates : DINT;
	nAxes :DINT;
	nOutputs :DINT;
	bInit : BOOL := FALSE;
	bAtState : BOOL;
	iAxis : DINT;
	stAxis : DUT_MotionStage;
	stState : DUT_PositionState;
	
	currState : DINT;
	nextState : DINT;
END_VAR

IF NOT bInit THEN
	bInit := TRUE;
	//nAssemblyStates := UPPER_BOUND(arrAssemblyStates, 1);
	nAssemblyStates := UPPER_BOUND(arrTransitions, 2); // take from # of columns in transition matrix
	nAxes := UPPER_BOUND(arrAxes, 1);
	nOutputs := UPPER_BOUND(arrOutputs, 1);
END_IF

// Determine current assembly state
currState := 0; // Start in the unknown state
FOR nextState := 1 TO nOutputs DO // For each defined output state
	bAtState := TRUE;
	FOR iAxis := 1 TO UPPER_BOUND(arrAxes,1) DO // check each axis for a match with the assembly position state
		bAtState := (bAtState AND F_AtPositionState(stMotionStage:=arrAxes[iAxis], stPositionState:=arrOutputs[nextState, iAxis]));
	END_FOR
	IF bAtState THEN
		currState := nextState;
	END_IF
END_FOR

// Reset logic before determining allowed moves
FOR nextState := 1 TO UPPER_BOUND(arrAssemblyStates, 1) DO
	FOR iAxis := 1 TO UPPER_BOUND(arrAxes, 1) DO
		arrOutputs[nextState, iAxis].bMoveOk := FALSE;
	END_FOR
END_FOR

// Update motion logic for next state based on current state
FOR nextState := 1 TO nAssemblyStates DO
	IF arrTransitions[currState, nextState] THEN
		FOR iAxis :=1 TO UPPER_BOUND(arrAxes, 1) DO
			arrOutputs[nextState, iAxis].bMoveOk := TRUE;
		END_FOR
	END_IF
END_FOR

END_FUNCTION_BLOCK

// ---- POUs/Assemblies/PRG_Illumination.TcPOU
PROGRAM PRG_Illumination
(*	Program for the ChemRIXS illumination system. *)
VAR_INPUT
	xMoveOK : BOOL := FALSE; // External interlock. Applied to bEnable of all PositionStateManagers.
END_VAR
VAR
	bInit : BOOL := FALSE; // Initialization variable
	
	// Motor axes

	stILMXMotor : DUT_MotionStage;

	stILMYMotor : DUT_MotionStage;
	stILMZMotor : DUT_MotionStage;
							
	// Define axis states for each axis. These are fed to a FB_PositionState manager for each axis
	// X axis position states
	stILMXPosPark : DUT_PositionState :=   (sName:= 'PARK',
										 	fPosition := 0.0,
										 	fDelta:=1.0,
									     	fVelocity:=5.0,
    									 	fAccel:=1.0, 
											fDecel:=1.0,
    									 	bMoveOk:=FALSE,
    									 	bLocked:=TRUE,
    									 	bValid:=TRUE);

	// Y axis position states
	stILMYPosPark : DUT_PositionState :=   (sName:= 'PARK',
										 	fPosition := 0.0,
										 	fDelta:=1.0,
									     	fVelocity:=5.0,
    									 	fAccel:=1.0, 
											fDecel:=1.0,
    									 	bMoveOk:=FALSE,
    									 	bLocked:=TRUE,
    									 	bValid:=TRUE);
											
	// Z axis position states						
	stILMZPosPark : DUT_PositionState :=   (sName:= 'PARK',
										 	fPosition := 0.0,
										 	fDelta:=1.0,
									     	fVelocity:=5.0,
    									 	fAccel:=1.0, 
											fDecel:=1.0,
    									 	bMoveOk:=FALSE,
    									 	bLocked:=TRUE,
    									 	bValid:=TRUE);
	
	fbILMXStage : FB_MotionStage;
	fbILMYStage : FB_MotionStage;
	fbILMZStage : FB_MotionStage;
	
END_VAR

fbILMXStage(stMotionStage := stILMXMotor);

END_PROGRAM

// ---- POUs/EPS/FB_BFS.TcPOU
FUNCTION_BLOCK FB_BFS
VAR_IN_OUT
	fbAdjacent : FB_AdjacentStates;
	arrTransitions: ARRAY [*, *] OF BOOL;
	arrAdjStates: ARRAY [*] OF ST_BFSAssemblyState;
	//arrAdjStates : ARRAY [*] OF DINT;
	nAdjacentStates : DINT;
	arrStates : ARRAY [*] OF ST_BFSAssemblyState;
	arrPath : ARRAY [*] OF ST_BFSAssemblyState;
	stQueue : ST_Queue;
	fbQueue : FB_Queue;
END_VAR
VAR_INPUT
	RootState : ST_BFSAssemblyState;
	Target : ST_BFSAssemblyState;
END_VAR
VAR_OUTPUT
	bError : BOOL; // an error occured, e.g. we didn't find the requested state
END_VAR
VAR
	Current : ST_BFSAssemblyState;
	Root	: ST_BFSAssemblyState;
	Adjacent : ST_BFSAssemblyState;
	iCounter : DINT;
	nStates : DINT;
	//
	iState : DINT;
	iTransition : DINT;
	bFound : BOOL := FALSE;
	Next : ST_BFSAssemblyState;
	iLower : DINT;
	iUpper : DINT;
	bFirst : BOOL;
END_VAR

THIS^.ClearStates();
Root := THIS^.GetState(iState:=RootState.iState, bDiscover:=TRUE); 
fbQueue.Enqueue(Root);
WHILE NOT fbQueue.Queue_Is_Empty() DO 
	Current := fbQueue.Dequeue(); 
	IF Current.iState = Target.iState THEN // found destination
		bFound := TRUE;
		EXIT;
	ELSE
		// Put adjacent states into arrAdjStates, count # of adjacent states
		THIS^.GetAdjacentStates(Current.iState); 
		// Mark any undiscovered states in arrAdjStates, add them to the queue, and label their parent state
		THIS^.DiscoverStates();
	END_IF
END_WHILE

// Stuff the target in first
//arrPath[1] := arrStates[Target.iState];
arrPath[1] := THIS^.GetState(iState:=Target.iState, bDiscover:=FALSE);
// Get the next state before starting loop
Current := THIS^.GetNextState(PrevState:=Target);
iCounter := 2;
WHILE Current.iParent <> 0 DO
	// Stuff state into path array
	arrPath[iCounter] := arrStates[Current.iState];
	// Locate the next child state
	Current := THIS^.GetNextState(PrevState:=Current);
	iCounter := iCounter + 1;
	IF iCounter >= nStates THEN
		EXIT; // Something bad happened. We exceeded the number of possible states.
	END_IF
END_WHILE

METHOD ClearStates : BOOL
VAR_INPUT
END_VAR
VAR
	Counter : DINT;
END_VAR
FOR Counter := LOWER_BOUND(arrStates,1) TO UPPER_BOUND(arrStates,1) DO // set all states to undiscovered, clear parent states
	arrStates[Counter].bDiscovered := FALSE;
	arrStates[Counter].iParent := 0;
END_FOR
END_METHOD

METHOD DiscoverStates : BOOL
VAR_INPUT
END_VAR
VAR
	Counter : DINT;
END_VAR
FOR Counter := LOWER_BOUND(arrAdjStates,1) TO nAdjacentStates DO // for all adjacent states
	Adjacent := arrAdjStates[Counter];
	IF NOT arrStates[Adjacent.iState].bDiscovered THEN // check that we haven't visited this one yet
		arrStates[Adjacent.iState].bDiscovered := TRUE; // mark state as discovered
		arrStates[Adjacent.iState].iParent := Current.iState;
		fbQueue.Enqueue(arrStates[Adjacent.iState]); // add state to queue to continue search
	END_IF
END_FOR
END_METHOD

METHOD GetAdjacentStates : BOOL
VAR_INPUT
	iStartState : DINT; // Node to expand find adjacent nodes from 
END_VAR
VAR
	stateCounter : DINT;
	transitionCounter : DINT;
END_VAR
transitionCounter := 0;
// Loop over all states to find states adjacent to the current state
FOR stateCounter := LOWER_BOUND(arrStates, 1) TO UPPER_BOUND(arrStates,1) DO // start at zero due to arrStates index
	iState := arrStates[stateCounter].iState; // pick out the state index of the state in question
	IF iState <> iStartState THEN // only look at transitions away from root state
		IF arrTransitions[iStartState, stateCounter] THEN // the transition is allowed
			transitionCounter := transitionCounter + 1;
			arrAdjStates[transitionCounter] := arrStates[stateCounter]; // save this adjacent state
		END_IF
	END_IF
END_FOR
nAdjacentStates := transitionCounter;
END_METHOD

METHOD GetNextState : ST_BFSAssemblyState
VAR_INPUT
	PrevState : ST_BFSAssemblyState;
END_VAR
VAR
	Counter : DINT;
END_VAR
// Find next state in path by following parent attribute
FOR Counter := LOWER_BOUND(arrStates, 1) TO UPPER_BOUND(arrStates, 1) DO
	IF PrevState.iParent = arrStates[Counter].iState THEN
		GetNextState := arrStates[Counter];
		EXIT;
	END_IF
END_FOR
END_METHOD

METHOD GetState : ST_BFSAssemblyState
VAR_INPUT
	iState : DINT;
	bDiscover : BOOL := FALSE; 
END_VAR
VAR
	Counter : DINT;
END_VAR
FOR Counter := LOWER_BOUND(arrStates,1) TO UPPER_BOUND(arrStates,1) DO
	IF arrStates[Counter].iState = iState THEN
		arrStates[Counter].bDiscovered := bDiscover; // set state to discovered
		GetState := arrStates[Counter];
	END_IF
END_FOR
END_METHOD

END_FUNCTION_BLOCK

// ---- POUs/EPS/FB_Queue.TcPOU
FUNCTION_BLOCK FB_Queue
VAR_INPUT
	stQ : ST_Queue;
END_VAR
VAR_OUTPUT
END_VAR
VAR
END_VAR

METHOD PUBLIC Dequeue : ST_BFSAssemblyState
VAR_INPUT
END_VAR
IF NOT THIS^.Queue_Is_Empty() THEN	
	Dequeue := stQ.arrQueue[stQ.iFront];
	stQ.iFront := stQ.iFront + 1;
	stQ.iCount := stQ.iCount - 1;
END_IF
END_METHOD

METHOD Empty_Queue : BOOL
VAR_INPUT
END_VAR
// Reset queue to ST_Queue initial values
stQ.iCount := 0;
stQ.iBack := -1;
stQ.iFront := 0;
END_METHOD

METHOD PUBLIC Enqueue : BOOL
VAR_INPUT
	element : ST_BFSAssemblyState;
END_VAR
IF 	NOT THIS^.Queue_Is_Full() THEN
	IF stQ.iBack = stQ.iLength THEN
		stQ.iBack := -1;
	END_IF
	stQ.iBack := stQ.iBack + 1;
	stQ.arrQueue[stQ.iBack] := element;
	stQ.iCount := stQ.iCount + 1;
	Enqueue := TRUE;
ELSE
	Enqueue := FALSE;
END_IF
END_METHOD

METHOD Queue_Is_Empty : BOOL
VAR_INPUT
END_VAR
IF stQ.iCount = 0 THEN
	Queue_Is_Empty := TRUE;
ELSE
	Queue_Is_Empty := FALSE;	
END_IF
END_METHOD

METHOD Queue_Is_Full : BOOL
VAR_INPUT
END_VAR
IF stQ.iCount = stQ.iLength THEN
	Queue_Is_Full := TRUE;
ELSE
	Queue_Is_Full := FALSE;
END_IF
END_METHOD

END_FUNCTION_BLOCK
